LIN {X 0,Y 392.441,Z 295.362,A -85,B 0,C 180,E1 -11714.837,E2 -11714.837} C_VEL
LIN {X 0,Y 393.126,Z 283.476,A -85,B 0,C 180,E1 -11715.821,E2 -11715.821} C_VEL
LIN {X 0,Y 393.865,Z 270.295,A -85,B 0,C 180,E1 -11716.664,E2 -11716.664} C_VEL
LIN {X 0,Y 392.022,Z 258.735,A -85,B 0,C 180,E1 -11717.291,E2 -11717.291} C_VEL
LIN {X 0,Y 389.995,Z 247.385,A -85,B 0,C 180,E1 -11717.777,E2 -11717.777} C_VEL
LIN {X 0,Y 390.225,Z 238.96,A -85,B 0,C 180,E1 -11721.113,E2 -11721.113} C_VEL
LIN {X 0,Y 390.437,Z 231.991,A -85,B 0,C 180,E1 -11723.891,E2 -11723.891} C_VEL
LIN {X 0,Y 390.676,Z 223.459,A -85,B 0,C 180,E1 -11727.305,E2 -11727.305} C_VEL
LIN {X 0,Y 391.018,Z 214.714,A -85,B 0,C 180,E1 -11730.825,E2 -11730.825} C_VEL
LIN {X 0,Y 391.238,Z 206.117,A -85,B 0,C 180,E1 -11734.276,E2 -11734.276} C_VEL
LIN {X 0,Y 391.129,Z 201.01,A -85,B 0,C 180,E1 -11736.368,E2 -11736.368} C_VEL
LIN {X 0,Y 390.133,Z 194.889,A -85,B 0,C 180,E1 -11739.004,E2 -11739.004} C_VEL
LIN {X 0,Y 390.044,Z 194.901,A -85,B 0,C 180,E1 -11742.373,E2 -11742.373} C_VEL
LIN {X 0,Y 390.049,Z 194.896,A -85,B 0,C 180,E1 -11745.354,E2 -11745.354} C_VEL
LIN {X 0,Y 390.036,Z 194.901,A -85,B 0,C 180,E1 -11748.186,E2 -11748.186} C_VEL
LIN {X 0,Y 390.07,Z 194.899,A -85,B 0,C 180,E1 -11750.904,E2 -11750.904} C_VEL
LIN {X 0,Y 390.073,Z 194.899,A -85,B 0,C 180,E1 -11754.791,E2 -11754.791} C_VEL
LIN {X 0,Y 390.025,Z 194.903,A -85,B 0,C 180,E1 -11757.878,E2 -11757.878} C_VEL
LIN {X 0,Y 389.947,Z 194.914,A -85,B 0,C 180,E1 -11759.895,E2 -11759.895} C_VEL
LIN {X 0,Y 389.913,Z 195.341,A -85,B 0,C 180,E1 -11760.877,E2 -11760.877} C_VEL
LIN {X 0,Y 389.906,Z 199.409,A -85,B 0,C 180,E1 -11764.366,E2 -11764.366} C_VEL
LIN {X 0,Y 389.783,Z 203.49,A -85,B 0,C 180,E1 -11767.749,E2 -11767.749} C_VEL
LIN {X 0,Y 389.715,Z 207.645,A -85,B 0,C 180,E1 -11771.057,E2 -11771.057} C_VEL
LIN {X 0,Y 389.681,Z 211.96,A -85,B 0,C 180,E1 -11774.303,E2 -11774.303} C_VEL
LIN {X 0,Y 389.761,Z 217.229,A -85,B 0,C 180,E1 -11777.965,E2 -11777.965} C_VEL
LIN {X 0,Y 392.368,Z 228.553,A -85,B 0,C 180,E1 -11778.57,E2 -11778.57} C_VEL
LIN {X 0,Y 393.371,Z 233.68,A -85,B 0,C 180,E1 -11778.926,E2 -11778.926} C_VEL
LIN {X 0,Y 393.133,Z 243.41,A -85,B 0,C 180,E1 -11779.701,E2 -11779.701} C_VEL
LIN {X 0,Y 392.736,Z 250.958,A -85,B 0,C 180,E1 -11780.516,E2 -11780.516} C_VEL
LIN {X 0,Y 392.364,Z 256.371,A -85,B 0,C 180,E1 -11781.241,E2 -11781.241} C_VEL
LIN {X 0,Y 391.909,Z 262.54,A -85,B 0,C 180,E1 -11782.269,E2 -11782.269} C_VEL
LIN {X 0,Y 391.395,Z 268.341,A -85,B 0,C 180,E1 -11783.555,E2 -11783.555} C_VEL
LIN {X 0,Y 391.078,Z 272.615,A -85,B 0,C 180,E1 -11784.843,E2 -11784.843} C_VEL
LIN {X 0,Y 390.802,Z 275.178,A -85,B 0,C 180,E1 -11785.874,E2 -11785.874} C_VEL
LIN {X 0,Y 390.417,Z 277.099,A -85,B 0,C 180,E1 -11786.903,E2 -11786.903} C_VEL
LIN {X 0,Y 390.359,Z 278.393,A -85,B 0,C 180,E1 -11787.935,E2 -11787.935} C_VEL
LIN {X 0,Y 390.23,Z 279.168,A -85,B 0,C 180,E1 -11788.967,E2 -11788.967} C_VEL
LIN {X 0,Y 390.176,Z 279.434,A -85,B 0,C 180,E1 -11789.999,E2 -11789.999} C_VEL
LIN {X 0,Y 390.225,Z 279.209,A -85,B 0,C 180,E1 -11791.031,E2 -11791.031} C_VEL
LIN {X 0,Y 390.346,Z 278.488,A -85,B 0,C 180,E1 -11792.062,E2 -11792.062} C_VEL
LIN {X 0,Y 390.412,Z 277.251,A -85,B 0,C 180,E1 -11793.094,E2 -11793.094} C_VEL
LIN {X 0,Y 390.993,Z 274.224,A -85,B 0,C 180,E1 -11794.638,E2 -11794.638} C_VEL
LIN {X 0,Y 391.149,Z 269.687,A -85,B 0,C 180,E1 -11796.187,E2 -11796.187} C_VEL
LIN {X 0,Y 391.589,Z 266.668,A -85,B 0,C 180,E1 -11796.957,E2 -11796.957} C_VEL
LIN {X 0,Y 391.858,Z 262.997,A -85,B 0,C 180,E1 -11797.729,E2 -11797.729} C_VEL
LIN {X 0,Y 392.281,Z 257.796,A -85,B 0,C 180,E1 -11798.638,E2 -11798.638} C_VEL
LIN {X 0,Y 392.719,Z 251.934,A -85,B 0,C 180,E1 -11799.46,E2 -11799.46} C_VEL
LIN {X 0,Y 392.996,Z 245.724,A -85,B 0,C 180,E1 -11800.165,E2 -11800.165} C_VEL
LIN {X 0,Y 393.411,Z 237.435,A -85,B 0,C 180,E1 -11800.901,E2 -11800.901} C_VEL
LIN {X 0,Y 393.293,Z 232.95,A -85,B 0,C 180,E1 -11801.227,E2 -11801.227} C_VEL
LIN {X 0,Y 391.615,Z 228.223,A -85,B 0,C 180,E1 -11801.632,E2 -11801.632} C_VEL
LIN {X 0,Y 388.24,Z 222.83,A -85,B 0,C 180,E1 -11802.267,E2 -11802.267} C_VEL
LIN {X 0,Y 384.867,Z 218.57,A -85,B 0,C 180,E1 -11803.042,E2 -11803.042} C_VEL
LIN {X 0,Y 383.099,Z 216.211,A -85,B 0,C 180,E1 -11803.745,E2 -11803.745} C_VEL
LIN {X 0,Y 382.664,Z 215.17,A -85,B 0,C 180,E1 -11804.269,E2 -11804.269} C_VEL
LIN {X 0,Y 382.713,Z 211.016,A -85,B 0,C 180,E1 -11807.27,E2 -11807.27} C_VEL
LIN {X 0,Y 382.734,Z 206.813,A -85,B 0,C 180,E1 -11810.528,E2 -11810.528} C_VEL
LIN {X 0,Y 382.798,Z 202.837,A -85,B 0,C 180,E1 -11813.821,E2 -11813.821} C_VEL
LIN {X 0,Y 382.902,Z 198.648,A -85,B 0,C 180,E1 -11817.312,E2 -11817.312} C_VEL
LIN {X 0,Y 382.853,Z 195.894,A -85,B 0,C 180,E1 -11819.71,E2 -11819.71} C_VEL
LIN {X 0,Y 382.976,Z 195.779,A -85,B 0,C 180,E1 -11822.419,E2 -11822.419} C_VEL
LIN {X 0,Y 383.022,Z 195.774,A -85,B 0,C 180,E1 -11825.954,E2 -11825.954} C_VEL
LIN {X 0,Y 383.01,Z 195.776,A -85,B 0,C 180,E1 -11829.585,E2 -11829.585} C_VEL
LIN {X 0,Y 382.999,Z 195.778,A -85,B 0,C 180,E1 -11832.777,E2 -11832.777} C_VEL
LIN {X 0,Y 382.991,Z 195.776,A -85,B 0,C 180,E1 -11835.788,E2 -11835.788} C_VEL
LIN {X 0,Y 382.982,Z 195.779,A -85,B 0,C 180,E1 -11838.794,E2 -11838.794} C_VEL
LIN {X 0,Y 382.994,Z 195.776,A -85,B 0,C 180,E1 -11842.094,E2 -11842.094} C_VEL
LIN {X 0,Y 383.01,Z 195.772,A -85,B 0,C 180,E1 -11845.331,E2 -11845.331} C_VEL
LIN {X 0,Y 383.028,Z 195.771,A -85,B 0,C 180,E1 -11847.852,E2 -11847.852} C_VEL
LIN {X 0,Y 383.054,Z 195.766,A -85,B 0,C 180,E1 -11851.719,E2 -11851.719} C_VEL
LIN {X 0,Y 383.042,Z 195.762,A -85,B 0,C 180,E1 -11855.039,E2 -11855.039} C_VEL
LIN {X 0,Y 382.983,Z 195.775,A -85,B 0,C 180,E1 -11858.468,E2 -11858.468} C_VEL
LIN {X 0,Y 383.079,Z 195.769,A -85,B 0,C 180,E1 -11861.827,E2 -11861.827} C_VEL
LIN {X 0,Y 383.102,Z 195.754,A -85,B 0,C 180,E1 -11865.118,E2 -11865.118} C_VEL
LIN {X 0,Y 383.087,Z 195.762,A -85,B 0,C 180,E1 -11868.358,E2 -11868.358} C_VEL
LIN {X 0,Y 383.252,Z 195.743,A -85,B 0,C 180,E1 -11871.976,E2 -11871.976} C_VEL
LIN {X 0,Y 383.185,Z 195.747,A -85,B 0,C 180,E1 -11874.738,E2 -11874.738} C_VEL
LIN {X 0,Y 383.376,Z 195.727,A -85,B 0,C 180,E1 -11877.899,E2 -11877.899} C_VEL
LIN {X 0,Y 383.507,Z 195.702,A -85,B 0,C 180,E1 -11880,E2 -11880} C_VEL
LIN {X 0,Y 383.231,Z 195.746,A -85,B 0,C 180,E1 -11883.154,E2 -11883.154} C_VEL
LIN {X 0,Y 383.272,Z 195.74,A -85,B 0,C 180,E1 -11886.316,E2 -11886.316} C_VEL
LIN {X 0,Y 383.248,Z 195.744,A -85,B 0,C 180,E1 -11888.436,E2 -11888.436} C_VEL
LIN {X 0,Y 383.124,Z 195.756,A -85,B 0,C 180,E1 -11892.716,E2 -11892.716} C_VEL
LIN {X 0,Y 383.069,Z 195.77,A -85,B 0,C 180,E1 -11895.974,E2 -11895.974} C_VEL
LIN {X 0,Y 383.047,Z 195.77,A -85,B 0,C 180,E1 -11899.284,E2 -11899.284} C_VEL
LIN {X 0,Y 382.977,Z 195.78,A -85,B 0,C 180,E1 -11902.667,E2 -11902.667} C_VEL
LIN {X 0,Y 382.971,Z 195.783,A -85,B 0,C 180,E1 -11906.131,E2 -11906.131} C_VEL
LIN {X 0,Y 382.965,Z 195.784,A -85,B 0,C 180,E1 -11909.702,E2 -11909.702} C_VEL
LIN {X 0,Y 382.993,Z 195.78,A -85,B 0,C 180,E1 -11913.402,E2 -11913.402} C_VEL
LIN {X 0,Y 383.021,Z 195.774,A -85,B 0,C 180,E1 -11916.165,E2 -11916.165} C_VEL
LIN {X 0,Y 382.967,Z 195.773,A -85,B 0,C 180,E1 -11919.964,E2 -11919.964} C_VEL
LIN {X 0,Y 382.997,Z 195.782,A -85,B 0,C 180,E1 -11922.78,E2 -11922.78} C_VEL
LIN {X 0,Y 382.99,Z 195.778,A -85,B 0,C 180,E1 -11925.791,E2 -11925.791} C_VEL
LIN {X 0,Y 383.02,Z 195.777,A -85,B 0,C 180,E1 -11929.572,E2 -11929.572} C_VEL
LIN {X 0,Y 384.924,Z 203.825,A -85,B 0,C 180,E1 -11932.293,E2 -11932.293} C_VEL
LIN {X 0,Y 387.231,Z 213.656,A -85,B 0,C 180,E1 -11935.321,E2 -11935.321} C_VEL
LIN {X 0,Y 389.234,Z 223.254,A -85,B 0,C 180,E1 -11938.063,E2 -11938.063} C_VEL
LIN {X 0,Y 389.391,Z 225.849,A -85,B 0,C 180,E1 -11938.743,E2 -11938.743} C_VEL
LIN {X 0,Y 387.181,Z 241.285,A -85,B 0,C 180,E1 -11942.488,E2 -11942.488} C_VEL
LIN {X 0,Y 385.301,Z 257.405,A -85,B 0,C 180,E1 -11946.343,E2 -11946.343} C_VEL
LIN {X 0,Y 383.784,Z 273.332,A -85,B 0,C 180,E1 -11950.199,E2 -11950.199} C_VEL
LIN {X 0,Y 383.267,Z 280.554,A -85,B 0,C 180,E1 -11951.977,E2 -11951.977} C_VEL
LIN {X 0,Y 385,Z 300.047,A -85,B 0,C 180,E1 -11952.636,E2 -11952.636} C_VEL
LIN {X 0,Y 385.65,Z 311.521,A -85,B 0,C 180,E1 -11953.185,E2 -11953.185} C_VEL
LIN {X 0,Y 385.742,Z 319.562,A -85,B 0,C 180,E1 -11953.666,E2 -11953.666} C_VEL
LIN {X 0,Y 384.928,Z 331.35,A -85,B 0,C 180,E1 -11954.514,E2 -11954.514} C_VEL
LIN {X 0,Y 384.273,Z 342.675,A -85,B 0,C 180,E1 -11955.559,E2 -11955.559} C_VEL
LIN {X 0,Y 383.547,Z 353.146,A -85,B 0,C 180,E1 -11956.761,E2 -11956.761} C_VEL
LIN {X 0,Y 382.946,Z 362.582,A -85,B 0,C 180,E1 -11958.086,E2 -11958.086} C_VEL
LIN {X 0,Y 382.337,Z 371.679,A -85,B 0,C 180,E1 -11959.677,E2 -11959.677} C_VEL
LIN {X 0,Y 382.054,Z 379.013,A -85,B 0,C 180,E1 -11961.272,E2 -11961.272} C_VEL
LIN {X 0,Y 381.91,Z 383.943,A -85,B 0,C 180,E1 -11962.6,E2 -11962.6} C_VEL
LIN {X 0,Y 381.775,Z 388.418,A -85,B 0,C 180,E1 -11964.093,E2 -11964.093} C_VEL
LIN {X 0,Y 381.786,Z 392.244,A -85,B 0,C 180,E1 -11965.779,E2 -11965.779} C_VEL
LIN {X 0,Y 381.861,Z 394.015,A -85,B 0,C 180,E1 -11966.836,E2 -11966.836} C_VEL
LIN {X 0,Y 381.878,Z 395.313,A -85,B 0,C 180,E1 -11967.892,E2 -11967.892} C_VEL
LIN {X 0,Y 381.878,Z 396.187,A -85,B 0,C 180,E1 -11968.947,E2 -11968.947} C_VEL
LIN {X 0,Y 381.914,Z 396.626,A -85,B 0,C 180,E1 -11970.001,E2 -11970.001} C_VEL
LIN {X 0,Y 381.857,Z 396.594,A -85,B 0,C 180,E1 -11971.056,E2 -11971.056} C_VEL
LIN {X 0,Y 381.866,Z 396.15,A -85,B 0,C 180,E1 -11972.111,E2 -11972.111} C_VEL
LIN {X 0,Y 381.779,Z 395.289,A -85,B 0,C 180,E1 -11973.167,E2 -11973.167} C_VEL
LIN {X 0,Y 381.77,Z 393.964,A -85,B 0,C 180,E1 -11974.224,E2 -11974.224} C_VEL
LIN {X 0,Y 381.77,Z 390.247,A -85,B 0,C 180,E1 -11976.233,E2 -11976.233} C_VEL
LIN {X 0,Y 381.983,Z 385.806,A -85,B 0,C 180,E1 -11977.933,E2 -11977.933} C_VEL
LIN {X 0,Y 382.401,Z 379.388,A -85,B 0,C 180,E1 -11979.789,E2 -11979.789} C_VEL
LIN {X 0,Y 382.931,Z 372.469,A -85,B 0,C 180,E1 -11981.38,E2 -11981.38} C_VEL
LIN {X 0,Y 383.876,Z 364.003,A -85,B 0,C 180,E1 -11982.961,E2 -11982.961} C_VEL
LIN {X 0,Y 384.806,Z 353.59,A -85,B 0,C 180,E1 -11984.538,E2 -11984.538} C_VEL
LIN {X 0,Y 386.105,Z 342.845,A -85,B 0,C 180,E1 -11985.846,E2 -11985.846} C_VEL
LIN {X 0,Y 387.472,Z 330.997,A -85,B 0,C 180,E1 -11987.008,E2 -11987.008} C_VEL
LIN {X 0,Y 388.687,Z 318.195,A -85,B 0,C 180,E1 -11988.011,E2 -11988.011} C_VEL
LIN {X 0,Y 388.737,Z 304.837,A -85,B 0,C 180,E1 -11988.892,E2 -11988.892} C_VEL
LIN {X 0,Y 387.598,Z 290.655,A -85,B 0,C 180,E1 -11989.68,E2 -11989.68} C_VEL
LIN {X 0,Y 385.077,Z 275.775,A -85,B 0,C 180,E1 -11990.475,E2 -11990.475} C_VEL
LIN {X 0,Y 384.394,Z 266.537,A -85,B 0,C 180,E1 -11991.45,E2 -11991.45} C_VEL
LIN {X 0,Y 386.367,Z 248.038,A -85,B 0,C 180,E1 -11995.886,E2 -11995.886} C_VEL
LIN {X 0,Y 388.604,Z 230.925,A -85,B 0,C 180,E1 -11999.996,E2 -11999.996} C_VEL
LIN {X 0,Y 389.414,Z 224.596,A -85,B 0,C 180,E1 -12001.561,E2 -12001.561} C_VEL
LIN {X 0,Y 387.476,Z 215.101,A -85,B 0,C 180,E1 -12004.214,E2 -12004.214} C_VEL
LIN {X 0,Y 385.15,Z 204.861,A -85,B 0,C 180,E1 -12007.354,E2 -12007.354} C_VEL
LIN {X 0,Y 384.083,Z 200.232,A -85,B 0,C 180,E1 -12008.887,E2 -12008.887} C_VEL
LIN {X 0,Y 384.548,Z 199.877,A -85,B 0,C 180,E1 -12009.862,E2 -12009.862} C_VEL
LIN {X 0,Y 384.84,Z 201.165,A -85,B 0,C 180,E1 -12013.073,E2 -12013.073} C_VEL
LIN {X 0,Y 385.222,Z 202.398,A -85,B 0,C 180,E1 -12014.641,E2 -12014.641} C_VEL
LIN {X 0,Y 386.114,Z 205.789,A -85,B 0,C 180,E1 -12017.665,E2 -12017.665} C_VEL
LIN {X 0,Y 387.063,Z 210.04,A -85,B 0,C 180,E1 -12020.543,E2 -12020.543} C_VEL
LIN {X 0,Y 387.815,Z 214.746,A -85,B 0,C 180,E1 -12023.271,E2 -12023.271} C_VEL
LIN {X 0,Y 387.943,Z 217.442,A -85,B 0,C 180,E1 -12024.611,E2 -12024.611} C_VEL
LIN {X 0,Y 386.832,Z 225.39,A -85,B 0,C 180,E1 -12028.205,E2 -12028.205} C_VEL
LIN {X 0,Y 386.084,Z 233.594,A -85,B 0,C 180,E1 -12031.752,E2 -12031.752} C_VEL
LIN {X 0,Y 385.508,Z 241.602,A -85,B 0,C 180,E1 -12035.209,E2 -12035.209} C_VEL
LIN {X 0,Y 384.943,Z 249.614,A -85,B 0,C 180,E1 -12038.612,E2 -12038.612} C_VEL
LIN {X 0,Y 384.852,Z 252.197,A -85,B 0,C 180,E1 -12039.664,E2 -12039.664} C_VEL
LIN {X 0,Y 389.3,Z 265.874,A -85,B 0,C 180,E1 -12040.724,E2 -12040.724} C_VEL
LIN {X 0,Y 391.121,Z 274.403,A -85,B 0,C 180,E1 -12041.405,E2 -12041.405} C_VEL
LIN {X 0,Y 390.072,Z 287.025,A -85,B 0,C 180,E1 -12042.3,E2 -12042.3} C_VEL
LIN {X 0,Y 388.872,Z 298.96,A -85,B 0,C 180,E1 -12043.372,E2 -12043.372} C_VEL
LIN {X 0,Y 387.61,Z 310.068,A -85,B 0,C 180,E1 -12044.623,E2 -12044.623} C_VEL
LIN {X 0,Y 386.508,Z 318.618,A -85,B 0,C 180,E1 -12045.79,E2 -12045.79} C_VEL
LIN {X 0,Y 385.488,Z 326.598,A -85,B 0,C 180,E1 -12047.095,E2 -12047.095} C_VEL
LIN {X 0,Y 384.521,Z 334.416,A -85,B 0,C 180,E1 -12048.669,E2 -12048.669} C_VEL
LIN {X 0,Y 383.62,Z 341.722,A -85,B 0,C 180,E1 -12050.51,E2 -12050.51} C_VEL
LIN {X 0,Y 382.899,Z 347.344,A -85,B 0,C 180,E1 -12052.38,E2 -12052.38} C_VEL
LIN {X 0,Y 382.407,Z 350.368,A -85,B 0,C 180,E1 -12053.669,E2 -12053.669} C_VEL
LIN {X 0,Y 382.386,Z 352.255,A -85,B 0,C 180,E1 -12054.727,E2 -12054.727} C_VEL
LIN {X 0,Y 382.246,Z 353.747,A -85,B 0,C 180,E1 -12055.782,E2 -12055.782} C_VEL
LIN {X 0,Y 382.043,Z 354.843,A -85,B 0,C 180,E1 -12056.836,E2 -12056.836} C_VEL
LIN {X 0,Y 381.887,Z 355.487,A -85,B 0,C 180,E1 -12057.891,E2 -12057.891} C_VEL
LIN {X 0,Y 381.777,Z 355.73,A -85,B 0,C 180,E1 -12058.945,E2 -12058.945} C_VEL
LIN {X 0,Y 381.725,Z 355.576,A -85,B 0,C 180,E1 -12060,E2 -12060} C_VEL
LIN {X 0,Y 381.742,Z 354.991,A -85,B 0,C 180,E1 -12061.055,E2 -12061.055} C_VEL
LIN {X 0,Y 381.827,Z 353.971,A -85,B 0,C 180,E1 -12062.11,E2 -12062.11} C_VEL
LIN {X 0,Y 381.878,Z 352.553,A -85,B 0,C 180,E1 -12063.165,E2 -12063.165} C_VEL
LIN {X 0,Y 381.921,Z 349.589,A -85,B 0,C 180,E1 -12064.75,E2 -12064.75} C_VEL
LIN {X 0,Y 382.122,Z 345.564,A -85,B 0,C 180,E1 -12066.336,E2 -12066.336} C_VEL
LIN {X 0,Y 382.464,Z 339.365,A -85,B 0,C 180,E1 -12068.187,E2 -12068.187} C_VEL
LIN {X 0,Y 382.954,Z 332.597,A -85,B 0,C 180,E1 -12069.774,E2 -12069.774} C_VEL
LIN {X 0,Y 383.495,Z 324.224,A -85,B 0,C 180,E1 -12071.362,E2 -12071.362} C_VEL
LIN {X 0,Y 384.135,Z 315.655,A -85,B 0,C 180,E1 -12072.683,E2 -12072.683} C_VEL
LIN {X 0,Y 384.915,Z 304.334,A -85,B 0,C 180,E1 -12074.11,E2 -12074.11} C_VEL
LIN {X 0,Y 385.671,Z 292.196,A -85,B 0,C 180,E1 -12075.321,E2 -12075.321} C_VEL
LIN {X 0,Y 386.335,Z 280.59,A -85,B 0,C 180,E1 -12076.242,E2 -12076.242} C_VEL
LIN {X 0,Y 386.905,Z 270.133,A -85,B 0,C 180,E1 -12076.896,E2 -12076.896} C_VEL
LIN {X 0,Y 384.444,Z 255.949,A -85,B 0,C 180,E1 -12077.653,E2 -12077.653} C_VEL
LIN {X 0,Y 382.945,Z 247.664,A -85,B 0,C 180,E1 -12078.024,E2 -12078.024} C_VEL
LIN {X 0,Y 383.22,Z 238.902,A -85,B 0,C 180,E1 -12081.518,E2 -12081.518} C_VEL
LIN {X 0,Y 383.427,Z 231.838,A -85,B 0,C 180,E1 -12084.357,E2 -12084.357} C_VEL
LIN {X 0,Y 383.696,Z 223.209,A -85,B 0,C 180,E1 -12087.845,E2 -12087.845} C_VEL
LIN {X 0,Y 384.063,Z 214.34,A -85,B 0,C 180,E1 -12091.435,E2 -12091.435} C_VEL
LIN {X 0,Y 384.305,Z 205.172,A -85,B 0,C 180,E1 -12095.173,E2 -12095.173} C_VEL
LIN {X 0,Y 383.848,Z 200.338,A -85,B 0,C 180,E1 -12097.172,E2 -12097.172} C_VEL
LIN {X 0,Y 383.08,Z 195.768,A -85,B 0,C 180,E1 -12099.183,E2 -12099.183} C_VEL
LIN {X 0,Y 383.011,Z 195.778,A -85,B 0,C 180,E1 -12102.778,E2 -12102.778} C_VEL
LIN {X 0,Y 383.003,Z 195.777,A -85,B 0,C 180,E1 -12105.789,E2 -12105.789} C_VEL
LIN {X 0,Y 382.993,Z 195.78,A -85,B 0,C 180,E1 -12108.795,E2 -12108.795} C_VEL
LIN {X 0,Y 383,Z 195.781,A -85,B 0,C 180,E1 -12112.097,E2 -12112.097} C_VEL
LIN {X 0,Y 383.016,Z 195.779,A -85,B 0,C 180,E1 -12115.331,E2 -12115.331} C_VEL
LIN {X 0,Y 383.004,Z 195.778,A -85,B 0,C 180,E1 -12117.849,E2 -12117.849} C_VEL
LIN {X 0,Y 382.856,Z 195.798,A -85,B 0,C 180,E1 -12120.287,E2 -12120.287} C_VEL
LIN {X 0,Y 382.913,Z 198.525,A -85,B 0,C 180,E1 -12122.686,E2 -12122.686} C_VEL
LIN {X 0,Y 382.8,Z 202.65,A -85,B 0,C 180,E1 -12126.176,E2 -12126.176} C_VEL
LIN {X 0,Y 382.739,Z 206.829,A -85,B 0,C 180,E1 -12129.58,E2 -12129.58} C_VEL
LIN {X 0,Y 382.717,Z 211.112,A -85,B 0,C 180,E1 -12132.912,E2 -12132.912} C_VEL
LIN {X 0,Y 382.717,Z 216.426,A -85,B 0,C 180,E1 -12136.722,E2 -12136.722} C_VEL
LIN {X 0,Y 382.771,Z 218,A -85,B 0,C 180,E1 -12137.708,E2 -12137.708} C_VEL
LIN {X 0,Y 385.092,Z 227.759,A -85,B 0,C 180,E1 -12138.218,E2 -12138.218} C_VEL
LIN {X 0,Y 386.503,Z 235.079,A -85,B 0,C 180,E1 -12138.727,E2 -12138.727} C_VEL
LIN {X 0,Y 386.249,Z 244.611,A -85,B 0,C 180,E1 -12139.515,E2 -12139.515} C_VEL
LIN {X 0,Y 385.828,Z 252.004,A -85,B 0,C 180,E1 -12140.334,E2 -12140.334} C_VEL
LIN {X 0,Y 385.435,Z 257.447,A -85,B 0,C 180,E1 -12141.083,E2 -12141.083} C_VEL
LIN {X 0,Y 384.947,Z 263.581,A -85,B 0,C 180,E1 -12142.129,E2 -12142.129} C_VEL
LIN {X 0,Y 384.417,Z 269.356,A -85,B 0,C 180,E1 -12143.438,E2 -12143.438} C_VEL
LIN {X 0,Y 384.082,Z 273.607,A -85,B 0,C 180,E1 -12144.749,E2 -12144.749} C_VEL
LIN {X 0,Y 383.799,Z 276.161,A -85,B 0,C 180,E1 -12145.798,E2 -12145.798} C_VEL
LIN {X 0,Y 383.403,Z 278.077,A -85,B 0,C 180,E1 -12146.846,E2 -12146.846} C_VEL
LIN {X 0,Y 383.34,Z 279.368,A -85,B 0,C 180,E1 -12147.897,E2 -12147.897} C_VEL
LIN {X 0,Y 383.206,Z 280.142,A -85,B 0,C 180,E1 -12148.948,E2 -12148.948} C_VEL
LIN {X 0,Y 383.15,Z 280.407,A -85,B 0,C 180,E1 -12149.999,E2 -12149.999} C_VEL
LIN {X 0,Y 383.201,Z 280.182,A -85,B 0,C 180,E1 -12151.05,E2 -12151.05} C_VEL
LIN {X 0,Y 383.327,Z 279.462,A -85,B 0,C 180,E1 -12152.1,E2 -12152.1} C_VEL
LIN {X 0,Y 383.398,Z 278.228,A -85,B 0,C 180,E1 -12153.151,E2 -12153.151} C_VEL
LIN {X 0,Y 383.995,Z 275.209,A -85,B 0,C 180,E1 -12154.723,E2 -12154.723} C_VEL
LIN {X 0,Y 384.163,Z 270.69,A -85,B 0,C 180,E1 -12156.3,E2 -12156.3} C_VEL
LIN {X 0,Y 384.617,Z 267.684,A -85,B 0,C 180,E1 -12157.084,E2 -12157.084} C_VEL
LIN {X 0,Y 384.901,Z 264.035,A -85,B 0,C 180,E1 -12157.87,E2 -12157.87} C_VEL
LIN {X 0,Y 385.423,Z 258.095,A -85,B 0,C 180,E1 -12158.915,E2 -12158.915} C_VEL
LIN {X 0,Y 385.908,Z 251.406,A -85,B 0,C 180,E1 -12159.842,E2 -12159.842} C_VEL
LIN {X 0,Y 386.288,Z 242.955,A -85,B 0,C 180,E1 -12160.746,E2 -12160.746} C_VEL
LIN {X 0,Y 386.512,Z 234.664,A -85,B 0,C 180,E1 -12161.403,E2 -12161.403} C_VEL
LIN {X 0,Y 384.452,Z 224.93,A -85,B 0,C 180,E1 -12162.05,E2 -12162.05} C_VEL
LIN {X 0,Y 382.738,Z 217.845,A -85,B 0,C 180,E1 -12162.425,E2 -12162.425} C_VEL
LIN {X 0,Y 382.664,Z 215.17,A -85,B 0,C 180,E1 -12164.269,E2 -12164.269} C_VEL
LIN {X 0,Y 381.98,Z 214.053,A -85,B 0,C 180,E1 -12165.131,E2 -12165.131} C_VEL
LIN {X 0,Y 379.149,Z 212.545,A -85,B 0,C 180,E1 -12166.543,E2 -12166.543} C_VEL
LIN {X 0,Y 376.766,Z 211.369,A -85,B 0,C 180,E1 -12167.686,E2 -12167.686} C_VEL
LIN {X 0,Y 375.744,Z 210.371,A -85,B 0,C 180,E1 -12168.566,E2 -12168.566} C_VEL
LIN {X 0,Y 375.659,Z 210.002,A -85,B 0,C 180,E1 -12168.863,E2 -12168.863} C_VEL
LIN {X 0,Y 375.729,Z 206.127,A -85,B 0,C 180,E1 -12171.967,E2 -12171.967} C_VEL
LIN {X 0,Y 375.78,Z 203.339,A -85,B 0,C 180,E1 -12174.294,E2 -12174.294} C_VEL
LIN {X 0,Y 375.858,Z 200.519,A -85,B 0,C 180,E1 -12176.663,E2 -12176.663} C_VEL
LIN {X 0,Y 375.855,Z 197.709,A -85,B 0,C 180,E1 -12179.087,E2 -12179.087} C_VEL
LIN {X 0,Y 375.888,Z 196.664,A -85,B 0,C 180,E1 -12180.317,E2 -12180.317} C_VEL
LIN {X 0,Y 375.943,Z 196.656,A -85,B 0,C 180,E1 -12182.827,E2 -12182.827} C_VEL
LIN {X 0,Y 375.954,Z 196.657,A -85,B 0,C 180,E1 -12185.414,E2 -12185.414} C_VEL
LIN {X 0,Y 375.97,Z 196.652,A -85,B 0,C 180,E1 -12188.269,E2 -12188.269} C_VEL
LIN {X 0,Y 375.929,Z 196.657,A -85,B 0,C 180,E1 -12191.599,E2 -12191.599} C_VEL
LIN {X 0,Y 375.947,Z 196.657,A -85,B 0,C 180,E1 -12195.263,E2 -12195.263} C_VEL
LIN {X 0,Y 375.934,Z 196.654,A -85,B 0,C 180,E1 -12199.132,E2 -12199.132} C_VEL
LIN {X 0,Y 375.959,Z 196.652,A -85,B 0,C 180,E1 -12201.911,E2 -12201.911} C_VEL
LIN {X 0,Y 375.971,Z 196.649,A -85,B 0,C 180,E1 -12205.331,E2 -12205.331} C_VEL
LIN {X 0,Y 375.968,Z 196.656,A -85,B 0,C 180,E1 -12208.439,E2 -12208.439} C_VEL
LIN {X 0,Y 375.993,Z 196.65,A -85,B 0,C 180,E1 -12212.141,E2 -12212.141} C_VEL
LIN {X 0,Y 375.996,Z 196.641,A -85,B 0,C 180,E1 -12214.538,E2 -12214.538} C_VEL
LIN {X 0,Y 375.953,Z 196.654,A -85,B 0,C 180,E1 -12218.045,E2 -12218.045} C_VEL
LIN {X 0,Y 376.013,Z 196.645,A -85,B 0,C 180,E1 -12221.473,E2 -12221.473} C_VEL
LIN {X 0,Y 376.05,Z 196.632,A -85,B 0,C 180,E1 -12224.832,E2 -12224.832} C_VEL
LIN {X 0,Y 376.039,Z 196.641,A -85,B 0,C 180,E1 -12228.136,E2 -12228.136} C_VEL
LIN {X 0,Y 376.207,Z 196.621,A -85,B 0,C 180,E1 -12231.919,E2 -12231.919} C_VEL
LIN {X 0,Y 376.157,Z 196.623,A -85,B 0,C 180,E1 -12234.64,E2 -12234.64} C_VEL
LIN {X 0,Y 376.342,Z 196.603,A -85,B 0,C 180,E1 -12237.86,E2 -12237.86} C_VEL
LIN {X 0,Y 376.477,Z 196.578,A -85,B 0,C 180,E1 -12240,E2 -12240} C_VEL
LIN {X 0,Y 376.17,Z 196.625,A -85,B 0,C 180,E1 -12243.213,E2 -12243.213} C_VEL
LIN {X 0,Y 376.232,Z 196.618,A -85,B 0,C 180,E1 -12246.435,E2 -12246.435} C_VEL
LIN {X 0,Y 376.194,Z 196.62,A -85,B 0,C 180,E1 -12248.595,E2 -12248.595} C_VEL
LIN {X 0,Y 376.037,Z 196.644,A -85,B 0,C 180,E1 -12251.864,E2 -12251.864} C_VEL
LIN {X 0,Y 376.046,Z 196.642,A -85,B 0,C 180,E1 -12255.168,E2 -12255.168} C_VEL
LIN {X 0,Y 375.991,Z 196.651,A -85,B 0,C 180,E1 -12258.528,E2 -12258.528} C_VEL
LIN {X 0,Y 375.943,Z 196.659,A -85,B 0,C 180,E1 -12261.956,E2 -12261.956} C_VEL
LIN {X 0,Y 375.947,Z 196.658,A -85,B 0,C 180,E1 -12264.285,E2 -12264.285} C_VEL
LIN {X 0,Y 375.906,Z 196.663,A -85,B 0,C 180,E1 -12267.866,E2 -12267.866} C_VEL
LIN {X 0,Y 375.947,Z 196.659,A -85,B 0,C 180,E1 -12271.563,E2 -12271.563} C_VEL
LIN {X 0,Y 375.947,Z 196.656,A -85,B 0,C 180,E1 -12275.417,E2 -12275.417} C_VEL
LIN {X 0,Y 375.927,Z 196.66,A -85,B 0,C 180,E1 -12278.264,E2 -12278.264} C_VEL
LIN {X 0,Y 375.911,Z 196.653,A -85,B 0,C 180,E1 -12281.599,E2 -12281.599} C_VEL
LIN {X 0,Y 375.919,Z 196.662,A -85,B 0,C 180,E1 -12284.733,E2 -12284.733} C_VEL
LIN {X 0,Y 375.927,Z 196.649,A -85,B 0,C 180,E1 -12288.401,E2 -12288.401} C_VEL
LIN {X 0,Y 375.972,Z 196.823,A -85,B 0,C 180,E1 -12289.065,E2 -12289.065} C_VEL
LIN {X 0,Y 377.751,Z 204.13,A -85,B 0,C 180,E1 -12291.622,E2 -12291.622} C_VEL
LIN {X 0,Y 380.267,Z 214.887,A -85,B 0,C 180,E1 -12295.047,E2 -12295.047} C_VEL
LIN {X 0,Y 382.452,Z 225.437,A -85,B 0,C 180,E1 -12298.11,E2 -12298.11} C_VEL
LIN {X 0,Y 382.237,Z 228.933,A -85,B 0,C 180,E1 -12299.016,E2 -12299.016} C_VEL
LIN {X 0,Y 379.837,Z 245.163,A -85,B 0,C 180,E1 -12303.046,E2 -12303.046} C_VEL
LIN {X 0,Y 378.066,Z 260.186,A -85,B 0,C 180,E1 -12306.734,E2 -12306.734} C_VEL
LIN {X 0,Y 376.56,Z 275.877,A -85,B 0,C 180,E1 -12310.655,E2 -12310.655} C_VEL
LIN {X 0,Y 376.226,Z 280.307,A -85,B 0,C 180,E1 -12311.74,E2 -12311.74} C_VEL
LIN {X 0,Y 377.957,Z 299.837,A -85,B 0,C 180,E1 -12312.42,E2 -12312.42} C_VEL
LIN {X 0,Y 378.62,Z 310.331,A -85,B 0,C 180,E1 -12312.933,E2 -12312.933} C_VEL
LIN {X 0,Y 378.752,Z 319.578,A -85,B 0,C 180,E1 -12313.495,E2 -12313.495} C_VEL
LIN {X 0,Y 377.919,Z 331.247,A -85,B 0,C 180,E1 -12314.358,E2 -12314.358} C_VEL
LIN {X 0,Y 377.186,Z 343.103,A -85,B 0,C 180,E1 -12315.488,E2 -12315.488} C_VEL
LIN {X 0,Y 376.456,Z 353.958,A -85,B 0,C 180,E1 -12316.781,E2 -12316.781} C_VEL
LIN {X 0,Y 375.826,Z 363.128,A -85,B 0,C 180,E1 -12318.131,E2 -12318.131} C_VEL
LIN {X 0,Y 375.234,Z 372.052,A -85,B 0,C 180,E1 -12319.752,E2 -12319.752} C_VEL
LIN {X 0,Y 374.961,Z 379.235,A -85,B 0,C 180,E1 -12321.378,E2 -12321.378} C_VEL
LIN {X 0,Y 374.79,Z 384.907,A -85,B 0,C 180,E1 -12323,E2 -12323} C_VEL
LIN {X 0,Y 374.758,Z 389.321,A -85,B 0,C 180,E1 -12324.621,E2 -12324.621} C_VEL
LIN {X 0,Y 374.715,Z 391.618,A -85,B 0,C 180,E1 -12325.699,E2 -12325.699} C_VEL
LIN {X 0,Y 374.765,Z 393.455,A -85,B 0,C 180,E1 -12326.776,E2 -12326.776} C_VEL
LIN {X 0,Y 374.809,Z 394.788,A -85,B 0,C 180,E1 -12327.852,E2 -12327.852} C_VEL
LIN {X 0,Y 374.801,Z 395.694,A -85,B 0,C 180,E1 -12328.927,E2 -12328.927} C_VEL
LIN {X 0,Y 374.833,Z 396.183,A -85,B 0,C 180,E1 -12330.001,E2 -12330.001} C_VEL
LIN {X 0,Y 374.782,Z 396.198,A -85,B 0,C 180,E1 -12331.076,E2 -12331.076} C_VEL
LIN {X 0,Y 374.794,Z 395.786,A -85,B 0,C 180,E1 -12332.151,E2 -12332.151} C_VEL
LIN {X 0,Y 374.679,Z 394.954,A -85,B 0,C 180,E1 -12333.227,E2 -12333.227} C_VEL
LIN {X 0,Y 374.689,Z 393.696,A -85,B 0,C 180,E1 -12334.304,E2 -12334.304} C_VEL
LIN {X 0,Y 374.688,Z 390.342,A -85,B 0,C 180,E1 -12336.216,E2 -12336.216} C_VEL
LIN {X 0,Y 374.91,Z 385.686,A -85,B 0,C 180,E1 -12338.084,E2 -12338.084} C_VEL
LIN {X 0,Y 375.371,Z 379.412,A -85,B 0,C 180,E1 -12339.974,E2 -12339.974} C_VEL
LIN {X 0,Y 376.098,Z 371.346,A -85,B 0,C 180,E1 -12341.863,E2 -12341.863} C_VEL
LIN {X 0,Y 376.956,Z 364.291,A -85,B 0,C 180,E1 -12343.204,E2 -12343.204} C_VEL
LIN {X 0,Y 377.903,Z 354.57,A -85,B 0,C 180,E1 -12344.745,E2 -12344.745} C_VEL
LIN {X 0,Y 379.337,Z 343.648,A -85,B 0,C 180,E1 -12346.137,E2 -12346.137} C_VEL
LIN {X 0,Y 380.764,Z 332.213,A -85,B 0,C 180,E1 -12347.317,E2 -12347.317} C_VEL
LIN {X 0,Y 382.124,Z 319.753,A -85,B 0,C 180,E1 -12348.347,E2 -12348.347} C_VEL
LIN {X 0,Y 382.388,Z 307.435,A -85,B 0,C 180,E1 -12349.218,E2 -12349.218} C_VEL
LIN {X 0,Y 381.453,Z 292.78,A -85,B 0,C 180,E1 -12350.104,E2 -12350.104} C_VEL
LIN {X 0,Y 379.099,Z 278.124,A -85,B 0,C 180,E1 -12350.926,E2 -12350.926} C_VEL
LIN {X 0,Y 378.518,Z 275.536,A -85,B 0,C 180,E1 -12351.09,E2 -12351.09} C_VEL
LIN {X 0,Y 377.757,Z 263.252,A -85,B 0,C 180,E1 -12352.493,E2 -12352.493} C_VEL
LIN {X 0,Y 379.708,Z 246.268,A -85,B 0,C 180,E1 -12356.669,E2 -12356.669} C_VEL
LIN {X 0,Y 382.237,Z 228.809,A -85,B 0,C 180,E1 -12360.987,E2 -12360.987} C_VEL
LIN {X 0,Y 382.43,Z 225.324,A -85,B 0,C 180,E1 -12361.895,E2 -12361.895} C_VEL
LIN {X 0,Y 380.241,Z 214.793,A -85,B 0,C 180,E1 -12364.959,E2 -12364.959} C_VEL
LIN {X 0,Y 377.981,Z 205.17,A -85,B 0,C 180,E1 -12368.034,E2 -12368.034} C_VEL
LIN {X 0,Y 378.508,Z 204.372,A -85,B 0,C 180,E1 -12369.147,E2 -12369.147} C_VEL
LIN {X 0,Y 378.75,Z 204.167,A -85,B 0,C 180,E1 -12370.502,E2 -12370.502} C_VEL
LIN {X 0,Y 379.122,Z 205.478,A -85,B 0,C 180,E1 -12373.7,E2 -12373.7} C_VEL
LIN {X 0,Y 379.726,Z 208.272,A -85,B 0,C 180,E1 -12376.78,E2 -12376.78} C_VEL
LIN {X 0,Y 380.532,Z 212.074,A -85,B 0,C 180,E1 -12379.728,E2 -12379.728} C_VEL
LIN {X 0,Y 381.22,Z 216.443,A -85,B 0,C 180,E1 -12382.528,E2 -12382.528} C_VEL
LIN {X 0,Y 381.415,Z 219.89,A -85,B 0,C 180,E1 -12384.422,E2 -12384.422} C_VEL
LIN {X 0,Y 380.365,Z 226.847,A -85,B 0,C 180,E1 -12387.6,E2 -12387.6} C_VEL
LIN {X 0,Y 379.507,Z 234.843,A -85,B 0,C 180,E1 -12391.217,E2 -12391.217} C_VEL
LIN {X 0,Y 378.684,Z 244.361,A -85,B 0,C 180,E1 -12395.423,E2 -12395.423} C_VEL
LIN {X 0,Y 378.064,Z 252.663,A -85,B 0,C 180,E1 -12399.015,E2 -12399.015} C_VEL
LIN {X 0,Y 382.423,Z 265.485,A -85,B 0,C 180,E1 -12400.085,E2 -12400.085} C_VEL
LIN {X 0,Y 384.688,Z 275.647,A -85,B 0,C 180,E1 -12400.948,E2 -12400.948} C_VEL
LIN {X 0,Y 384.441,Z 280.567,A -85,B 0,C 180,E1 -12401.295,E2 -12401.295} C_VEL
LIN {X 0,Y 383.202,Z 292.877,A -85,B 0,C 180,E1 -12402.289,E2 -12402.289} C_VEL
LIN {X 0,Y 381.906,Z 303.782,A -85,B 0,C 180,E1 -12403.381,E2 -12403.381} C_VEL
LIN {X 0,Y 380.486,Z 314.649,A -85,B 0,C 180,E1 -12404.739,E2 -12404.739} C_VEL
LIN {X 0,Y 379.253,Z 323.345,A -85,B 0,C 180,E1 -12406.06,E2 -12406.06} C_VEL
LIN {X 0,Y 378.073,Z 331.855,A -85,B 0,C 180,E1 -12407.656,E2 -12407.656} C_VEL
LIN {X 0,Y 377.239,Z 338.755,A -85,B 0,C 180,E1 -12409.263,E2 -12409.263} C_VEL
LIN {X 0,Y 376.426,Z 344.339,A -85,B 0,C 180,E1 -12410.869,E2 -12410.869} C_VEL
LIN {X 0,Y 375.852,Z 348.728,A -85,B 0,C 180,E1 -12412.479,E2 -12412.479} C_VEL
LIN {X 0,Y 375.39,Z 351.06,A -85,B 0,C 180,E1 -12413.55,E2 -12413.55} C_VEL
LIN {X 0,Y 375.339,Z 352.898,A -85,B 0,C 180,E1 -12414.628,E2 -12414.628} C_VEL
LIN {X 0,Y 375.207,Z 354.342,A -85,B 0,C 180,E1 -12415.703,E2 -12415.703} C_VEL
LIN {X 0,Y 374.993,Z 355.372,A -85,B 0,C 180,E1 -12416.777,E2 -12416.777} C_VEL
LIN {X 0,Y 374.824,Z 355.966,A -85,B 0,C 180,E1 -12417.851,E2 -12417.851} C_VEL
LIN {X 0,Y 374.708,Z 356.167,A -85,B 0,C 180,E1 -12418.925,E2 -12418.925} C_VEL
LIN {X 0,Y 374.655,Z 355.964,A -85,B 0,C 180,E1 -12420,E2 -12420} C_VEL
LIN {X 0,Y 374.674,Z 355.308,A -85,B 0,C 180,E1 -12421.075,E2 -12421.075} C_VEL
LIN {X 0,Y 374.746,Z 354.246,A -85,B 0,C 180,E1 -12422.15,E2 -12422.15} C_VEL
LIN {X 0,Y 374.783,Z 352.785,A -85,B 0,C 180,E1 -12423.225,E2 -12423.225} C_VEL
LIN {X 0,Y 374.86,Z 349.734,A -85,B 0,C 180,E1 -12424.84,E2 -12424.84} C_VEL
LIN {X 0,Y 375.092,Z 344.712,A -85,B 0,C 180,E1 -12426.753,E2 -12426.753} C_VEL
LIN {X 0,Y 375.471,Z 338.254,A -85,B 0,C 180,E1 -12428.612,E2 -12428.612} C_VEL
LIN {X 0,Y 375.984,Z 331.113,A -85,B 0,C 180,E1 -12430.229,E2 -12430.229} C_VEL
LIN {X 0,Y 376.587,Z 322.251,A -85,B 0,C 180,E1 -12431.846,E2 -12431.846} C_VEL
LIN {X 0,Y 377.411,Z 312.233,A -85,B 0,C 180,E1 -12433.323,E2 -12433.323} C_VEL
LIN {X 0,Y 378.142,Z 301.58,A -85,B 0,C 180,E1 -12434.596,E2 -12434.596} C_VEL
LIN {X 0,Y 378.763,Z 291.247,A -85,B 0,C 180,E1 -12435.608,E2 -12435.608} C_VEL
LIN {X 0,Y 379.469,Z 279.237,A -85,B 0,C 180,E1 -12436.544,E2 -12436.544} C_VEL
LIN {X 0,Y 379.898,Z 270.801,A -85,B 0,C 180,E1 -12437.079,E2 -12437.079} C_VEL
LIN {X 0,Y 377.515,Z 257.003,A -85,B 0,C 180,E1 -12437.842,E2 -12437.842} C_VEL
LIN {X 0,Y 375.907,Z 247.998,A -85,B 0,C 180,E1 -12438.248,E2 -12438.248} C_VEL
LIN {X 0,Y 376.21,Z 238.821,A -85,B 0,C 180,E1 -12441.939,E2 -12441.939} C_VEL
LIN {X 0,Y 376.437,Z 231.664,A -85,B 0,C 180,E1 -12444.839,E2 -12444.839} C_VEL
LIN {X 0,Y 376.708,Z 223.236,A -85,B 0,C 180,E1 -12448.275,E2 -12448.275} C_VEL
LIN {X 0,Y 377.091,Z 213.93,A -85,B 0,C 180,E1 -12452.085,E2 -12452.085} C_VEL
LIN {X 0,Y 377.285,Z 206.12,A -85,B 0,C 180,E1 -12455.273,E2 -12455.273} C_VEL
LIN {X 0,Y 376.802,Z 201.274,A -85,B 0,C 180,E1 -12457.313,E2 -12457.313} C_VEL
LIN {X 0,Y 376.014,Z 196.648,A -85,B 0,C 180,E1 -12459.383,E2 -12459.383} C_VEL
LIN {X 0,Y 375.939,Z 196.657,A -85,B 0,C 180,E1 -12463.189,E2 -12463.189} C_VEL
LIN {X 0,Y 375.94,Z 196.656,A -85,B 0,C 180,E1 -12466.81,E2 -12466.81} C_VEL
LIN {X 0,Y 375.952,Z 196.658,A -85,B 0,C 180,E1 -12470.535,E2 -12470.535} C_VEL
LIN {X 0,Y 375.962,Z 196.658,A -85,B 0,C 180,E1 -12473.496,E2 -12473.496} C_VEL
LIN {X 0,Y 375.962,Z 196.657,A -85,B 0,C 180,E1 -12475.887,E2 -12475.887} C_VEL
LIN {X 0,Y 375.879,Z 196.667,A -85,B 0,C 180,E1 -12479.327,E2 -12479.327} C_VEL
LIN {X 0,Y 375.896,Z 196.665,A -85,B 0,C 180,E1 -12479.68,E2 -12479.68} C_VEL
LIN {X 0,Y 375.895,Z 198.211,A -85,B 0,C 180,E1 -12481.492,E2 -12481.492} C_VEL
LIN {X 0,Y 375.839,Z 201.765,A -85,B 0,C 180,E1 -12484.526,E2 -12484.526} C_VEL
LIN {X 0,Y 375.784,Z 204.542,A -85,B 0,C 180,E1 -12486.873,E2 -12486.873} C_VEL
LIN {X 0,Y 375.679,Z 208.813,A -85,B 0,C 180,E1 -12490.321,E2 -12490.321} C_VEL
LIN {X 0,Y 375.695,Z 211.738,A -85,B 0,C 180,E1 -12492.583,E2 -12492.583} C_VEL
LIN {X 0,Y 375.711,Z 217.277,A -85,B 0,C 180,E1 -12496.584,E2 -12496.584} C_VEL
LIN {X 0,Y 375.768,Z 218.705,A -85,B 0,C 180,E1 -12497.424,E2 -12497.424} C_VEL
LIN {X 0,Y 378.067,Z 228.16,A -85,B 0,C 180,E1 -12497.927,E2 -12497.927} C_VEL
LIN {X 0,Y 379.643,Z 236.474,A -85,B 0,C 180,E1 -12498.52,E2 -12498.52} C_VEL
LIN {X 0,Y 379.36,Z 245.803,A -85,B 0,C 180,E1 -12499.322,E2 -12499.322} C_VEL
LIN {X 0,Y 378.921,Z 253.079,A -85,B 0,C 180,E1 -12500.15,E2 -12500.15} C_VEL
LIN {X 0,Y 378.508,Z 258.522,A -85,B 0,C 180,E1 -12500.918,E2 -12500.918} C_VEL
LIN {X 0,Y 377.988,Z 264.617,A -85,B 0,C 180,E1 -12501.983,E2 -12501.983} C_VEL
LIN {X 0,Y 377.425,Z 270.37,A -85,B 0,C 180,E1 -12503.315,E2 -12503.315} C_VEL
LIN {X 0,Y 377.087,Z 274.599,A -85,B 0,C 180,E1 -12504.652,E2 -12504.652} C_VEL
LIN {X 0,Y 376.797,Z 277.144,A -85,B 0,C 180,E1 -12505.72,E2 -12505.72} C_VEL
LIN {X 0,Y 376.389,Z 279.055,A -85,B 0,C 180,E1 -12506.787,E2 -12506.787} C_VEL
LIN {X 0,Y 376.32,Z 280.342,A -85,B 0,C 180,E1 -12507.858,E2 -12507.858} C_VEL
LIN {X 0,Y 376.182,Z 281.116,A -85,B 0,C 180,E1 -12508.928,E2 -12508.928} C_VEL
LIN {X 0,Y 376.124,Z 281.381,A -85,B 0,C 180,E1 -12509.999,E2 -12509.999} C_VEL
LIN {X 0,Y 376.177,Z 281.156,A -85,B 0,C 180,E1 -12511.069,E2 -12511.069} C_VEL
LIN {X 0,Y 376.309,Z 280.436,A -85,B 0,C 180,E1 -12512.139,E2 -12512.139} C_VEL
LIN {X 0,Y 376.385,Z 279.205,A -85,B 0,C 180,E1 -12513.21,E2 -12513.21} C_VEL
LIN {X 0,Y 376.996,Z 276.193,A -85,B 0,C 180,E1 -12514.811,E2 -12514.811} C_VEL
LIN {X 0,Y 377.178,Z 271.691,A -85,B 0,C 180,E1 -12516.418,E2 -12516.418} C_VEL
LIN {X 0,Y 377.646,Z 268.698,A -85,B 0,C 180,E1 -12517.215,E2 -12517.215} C_VEL
LIN {X 0,Y 377.943,Z 265.073,A -85,B 0,C 180,E1 -12518.015,E2 -12518.015} C_VEL
LIN {X 0,Y 378.498,Z 259.163,A -85,B 0,C 180,E1 -12519.079,E2 -12519.079} C_VEL
LIN {X 0,Y 379.013,Z 252.44,A -85,B 0,C 180,E1 -12520.034,E2 -12520.034} C_VEL
LIN {X 0,Y 379.419,Z 243.905,A -85,B 0,C 180,E1 -12520.97,E2 -12520.97} C_VEL
LIN {X 0,Y 379.673,Z 236.044,A -85,B 0,C 180,E1 -12521.612,E2 -12521.612} C_VEL
LIN {X 0,Y 377.651,Z 226.295,A -85,B 0,C 180,E1 -12522.288,E2 -12522.288} C_VEL
LIN {X 0,Y 375.726,Z 218.493,A -85,B 0,C 180,E1 -12522.695,E2 -12522.695} C_VEL
LIN {X 0,Y 375.644,Z 213.392,A -85,B 0,C 180,E1 -12526.297,E2 -12526.297} C_VEL
LIN {X 0,Y 375.659,Z 210.002,A -85,B 0,C 180,E1 -12528.863,E2 -12528.863} C_VEL
LIN {X 0,Y 374.987,Z 208.992,A -85,B 0,C 180,E1 -12529.744,E2 -12529.744} C_VEL
LIN {X 0,Y 372.148,Z 207.618,A -85,B 0,C 180,E1 -12531.186,E2 -12531.186} C_VEL
LIN {X 0,Y 369.789,Z 206.577,A -85,B 0,C 180,E1 -12532.353,E2 -12532.353} C_VEL
LIN {X 0,Y 368.831,Z 205.662,A -85,B 0,C 180,E1 -12533.252,E2 -12533.252} C_VEL
LIN {X 0,Y 368.782,Z 205.316,A -85,B 0,C 180,E1 -12533.555,E2 -12533.555} C_VEL
LIN {X 0,Y 368.848,Z 201.003,A -85,B 0,C 180,E1 -12537.211,E2 -12537.211} C_VEL
LIN {X 0,Y 368.842,Z 197.542,A -85,B 0,C 180,E1 -12540.325,E2 -12540.325} C_VEL
LIN {X 0,Y 368.891,Z 197.537,A -85,B 0,C 180,E1 -12543.537,E2 -12543.537} C_VEL
LIN {X 0,Y 368.898,Z 197.533,A -85,B 0,C 180,E1 -12546.855,E2 -12546.855} C_VEL
LIN {X 0,Y 368.906,Z 197.532,A -85,B 0,C 180,E1 -12550.369,E2 -12550.369} C_VEL
LIN {X 0,Y 368.877,Z 197.533,A -85,B 0,C 180,E1 -12553.615,E2 -12553.615} C_VEL
LIN {X 0,Y 368.878,Z 197.534,A -85,B 0,C 180,E1 -12556.694,E2 -12556.694} C_VEL
LIN {X 0,Y 368.905,Z 197.528,A -85,B 0,C 180,E1 -12559.641,E2 -12559.641} C_VEL
LIN {X 0,Y 368.895,Z 197.532,A -85,B 0,C 180,E1 -12563.143,E2 -12563.143} C_VEL
LIN {X 0,Y 368.892,Z 197.53,A -85,B 0,C 180,E1 -12566.461,E2 -12566.461} C_VEL
LIN {X 0,Y 368.915,Z 197.526,A -85,B 0,C 180,E1 -12570.309,E2 -12570.309} C_VEL
LIN {X 0,Y 368.972,Z 197.523,A -85,B 0,C 180,E1 -12573.534,E2 -12573.534} C_VEL
LIN {X 0,Y 368.956,Z 197.527,A -85,B 0,C 180,E1 -12576.421,E2 -12576.421} C_VEL
LIN {X 0,Y 368.926,Z 197.523,A -85,B 0,C 180,E1 -12579.946,E2 -12579.946} C_VEL
LIN {X 0,Y 368.968,Z 197.525,A -85,B 0,C 180,E1 -12583.398,E2 -12583.398} C_VEL
LIN {X 0,Y 369.047,Z 197.512,A -85,B 0,C 180,E1 -12586.79,E2 -12586.79} C_VEL
LIN {X 0,Y 369.057,Z 197.503,A -85,B 0,C 180,E1 -12590.131,E2 -12590.131} C_VEL
LIN {X 0,Y 369.187,Z 197.495,A -85,B 0,C 180,E1 -12593.441,E2 -12593.441} C_VEL
LIN {X 0,Y 369.307,Z 197.48,A -85,B 0,C 180,E1 -12597.819,E2 -12597.819} C_VEL
LIN {X 0,Y 369.446,Z 197.453,A -85,B 0,C 180,E1 -12600,E2 -12600} C_VEL
LIN {X 0,Y 369.303,Z 197.48,A -85,B 0,C 180,E1 -12602.181,E2 -12602.181} C_VEL
LIN {X 0,Y 369.194,Z 197.496,A -85,B 0,C 180,E1 -12606.558,E2 -12606.558} C_VEL
LIN {X 0,Y 369.126,Z 197.499,A -85,B 0,C 180,E1 -12608.761,E2 -12608.761} C_VEL
LIN {X 0,Y 368.993,Z 197.523,A -85,B 0,C 180,E1 -12612.094,E2 -12612.094} C_VEL
LIN {X 0,Y 368.985,Z 197.522,A -85,B 0,C 180,E1 -12615.465,E2 -12615.465} C_VEL
LIN {X 0,Y 368.942,Z 197.527,A -85,B 0,C 180,E1 -12618.895,E2 -12618.895} C_VEL
LIN {X 0,Y 368.908,Z 197.534,A -85,B 0,C 180,E1 -12622.397,E2 -12622.397} C_VEL
LIN {X 0,Y 368.908,Z 197.535,A -85,B 0,C 180,E1 -12625.987,E2 -12625.987} C_VEL
LIN {X 0,Y 368.882,Z 197.538,A -85,B 0,C 180,E1 -12629.693,E2 -12629.693} C_VEL
LIN {X 0,Y 368.887,Z 197.535,A -85,B 0,C 180,E1 -12633.044,E2 -12633.044} C_VEL
LIN {X 0,Y 368.907,Z 197.533,A -85,B 0,C 180,E1 -12636.198,E2 -12636.198} C_VEL
LIN {X 0,Y 368.866,Z 197.54,A -85,B 0,C 180,E1 -12638.958,E2 -12638.958} C_VEL
LIN {X 0,Y 368.863,Z 197.536,A -85,B 0,C 180,E1 -12642.009,E2 -12642.009} C_VEL
LIN {X 0,Y 368.872,Z 197.536,A -85,B 0,C 180,E1 -12645.177,E2 -12645.177} C_VEL
LIN {X 0,Y 368.911,Z 197.644,A -85,B 0,C 180,E1 -12648.472,E2 -12648.472} C_VEL
LIN {X 0,Y 371.094,Z 206.642,A -85,B 0,C 180,E1 -12651.665,E2 -12651.665} C_VEL
LIN {X 0,Y 373.709,Z 217.953,A -85,B 0,C 180,E1 -12655.33,E2 -12655.33} C_VEL
LIN {X 0,Y 375.503,Z 226.76,A -85,B 0,C 180,E1 -12657.937,E2 -12657.937} C_VEL
LIN {X 0,Y 375.445,Z 229.592,A -85,B 0,C 180,E1 -12658.706,E2 -12658.706} C_VEL
LIN {X 0,Y 373.009,Z 245.175,A -85,B 0,C 180,E1 -12662.674,E2 -12662.674} C_VEL
LIN {X 0,Y 371.063,Z 260.628,A -85,B 0,C 180,E1 -12666.565,E2 -12666.565} C_VEL
LIN {X 0,Y 369.508,Z 276.178,A -85,B 0,C 180,E1 -12670.56,E2 -12670.56} C_VEL
LIN {X 0,Y 369.183,Z 279.7,A -85,B 0,C 180,E1 -12671.486,E2 -12671.486} C_VEL
LIN {X 0,Y 370.922,Z 299.473,A -85,B 0,C 180,E1 -12672.196,E2 -12672.196} C_VEL
LIN {X 0,Y 371.655,Z 311.654,A -85,B 0,C 180,E1 -12672.816,E2 -12672.816} C_VEL
LIN {X 0,Y 371.632,Z 320.483,A -85,B 0,C 180,E1 -12673.381,E2 -12673.381} C_VEL
LIN {X 0,Y 370.912,Z 331.074,A -85,B 0,C 180,E1 -12674.196,E2 -12674.196} C_VEL
LIN {X 0,Y 370.227,Z 342.366,A -85,B 0,C 180,E1 -12675.293,E2 -12675.293} C_VEL
LIN {X 0,Y 369.434,Z 352.836,A -85,B 0,C 180,E1 -12676.555,E2 -12676.555} C_VEL
LIN {X 0,Y 368.831,Z 361.991,A -85,B 0,C 180,E1 -12677.902,E2 -12677.902} C_VEL
LIN {X 0,Y 368.19,Z 371.033,A -85,B 0,C 180,E1 -12679.554,E2 -12679.554} C_VEL
LIN {X 0,Y 367.887,Z 378.333,A -85,B 0,C 180,E1 -12681.211,E2 -12681.211} C_VEL
LIN {X 0,Y 367.732,Z 384.132,A -85,B 0,C 180,E1 -12682.865,E2 -12682.865} C_VEL
LIN {X 0,Y 367.663,Z 388.626,A -85,B 0,C 180,E1 -12684.517,E2 -12684.517} C_VEL
LIN {X 0,Y 367.646,Z 390.965,A -85,B 0,C 180,E1 -12685.616,E2 -12685.616} C_VEL
LIN {X 0,Y 367.673,Z 392.852,A -85,B 0,C 180,E1 -12686.714,E2 -12686.714} C_VEL
LIN {X 0,Y 367.741,Z 394.252,A -85,B 0,C 180,E1 -12687.811,E2 -12687.811} C_VEL
LIN {X 0,Y 367.728,Z 395.192,A -85,B 0,C 180,E1 -12688.906,E2 -12688.906} C_VEL
LIN {X 0,Y 367.754,Z 395.716,A -85,B 0,C 180,E1 -12690.001,E2 -12690.001} C_VEL
LIN {X 0,Y 367.709,Z 395.801,A -85,B 0,C 180,E1 -12691.097,E2 -12691.097} C_VEL
LIN {X 0,Y 367.704,Z 395.424,A -85,B 0,C 180,E1 -12692.192,E2 -12692.192} C_VEL
LIN {X 0,Y 367.584,Z 394.626,A -85,B 0,C 180,E1 -12693.29,E2 -12693.29} C_VEL
LIN {X 0,Y 367.61,Z 393.423,A -85,B 0,C 180,E1 -12694.387,E2 -12694.387} C_VEL
LIN {X 0,Y 367.586,Z 390.514,A -85,B 0,C 180,E1 -12696.169,E2 -12696.169} C_VEL
LIN {X 0,Y 367.859,Z 385.594,A -85,B 0,C 180,E1 -12698.24,E2 -12698.24} C_VEL
LIN {X 0,Y 368.254,Z 380.43,A -85,B 0,C 180,E1 -12699.892,E2 -12699.892} C_VEL
LIN {X 0,Y 368.855,Z 374.001,A -85,B 0,C 180,E1 -12701.542,E2 -12701.542} C_VEL
LIN {X 0,Y 369.91,Z 366.123,A -85,B 0,C 180,E1 -12703.18,E2 -12703.18} C_VEL
LIN {X 0,Y 370.92,Z 356.286,A -85,B 0,C 180,E1 -12704.853,E2 -12704.853} C_VEL
LIN {X 0,Y 372.3,Z 346.743,A -85,B 0,C 180,E1 -12706.168,E2 -12706.168} C_VEL
LIN {X 0,Y 373.88,Z 334.818,A -85,B 0,C 180,E1 -12707.504,E2 -12707.504} C_VEL
LIN {X 0,Y 375.392,Z 323.114,A -85,B 0,C 180,E1 -12708.56,E2 -12708.56} C_VEL
LIN {X 0,Y 376.015,Z 308.516,A -85,B 0,C 180,E1 -12709.661,E2 -12709.661} C_VEL
LIN {X 0,Y 375.299,Z 294.609,A -85,B 0,C 180,E1 -12710.557,E2 -12710.557} C_VEL
LIN {X 0,Y 373.218,Z 280.677,A -85,B 0,C 180,E1 -12711.39,E2 -12711.39} C_VEL
LIN {X 0,Y 372.075,Z 274.665,A -85,B 0,C 180,E1 -12711.802,E2 -12711.802} C_VEL
LIN {X 0,Y 371.295,Z 262.858,A -85,B 0,C 180,E1 -12713.275,E2 -12713.275} C_VEL
LIN {X 0,Y 371.228,Z 259.143,A -85,B 0,C 180,E1 -12713.797,E2 -12713.797} C_VEL
LIN {X 0,Y 373.249,Z 243.457,A -85,B 0,C 180,E1 -12717.751,E2 -12717.751} C_VEL
LIN {X 0,Y 375.572,Z 228.313,A -85,B 0,C 180,E1 -12721.599,E2 -12721.599} C_VEL
LIN {X 0,Y 374.879,Z 223.674,A -85,B 0,C 180,E1 -12722.935,E2 -12722.935} C_VEL
LIN {X 0,Y 372.786,Z 214.112,A -85,B 0,C 180,E1 -12725.839,E2 -12725.839} C_VEL
LIN {X 0,Y 371.971,Z 210.612,A -85,B 0,C 180,E1 -12727.032,E2 -12727.032} C_VEL
LIN {X 0,Y 372.878,Z 208.582,A -85,B 0,C 180,E1 -12729.397,E2 -12729.397} C_VEL
LIN {X 0,Y 372.953,Z 208.486,A -85,B 0,C 180,E1 -12731.267,E2 -12731.267} C_VEL
LIN {X 0,Y 373.212,Z 209.826,A -85,B 0,C 180,E1 -12734.309,E2 -12734.309} C_VEL
LIN {X 0,Y 373.758,Z 212.602,A -85,B 0,C 180,E1 -12737.396,E2 -12737.396} C_VEL
LIN {X 0,Y 374.409,Z 216.306,A -85,B 0,C 180,E1 -12740.341,E2 -12740.341} C_VEL
LIN {X 0,Y 374.918,Z 220.598,A -85,B 0,C 180,E1 -12743.14,E2 -12743.14} C_VEL
LIN {X 0,Y 374.927,Z 223.1,A -85,B 0,C 180,E1 -12744.472,E2 -12744.472} C_VEL
LIN {X 0,Y 373.404,Z 232.258,A -85,B 0,C 180,E1 -12748.829,E2 -12748.829} C_VEL
LIN {X 0,Y 372.514,Z 240.144,A -85,B 0,C 180,E1 -12752.466,E2 -12752.466} C_VEL
LIN {X 0,Y 371.813,Z 248.033,A -85,B 0,C 180,E1 -12756.022,E2 -12756.022} C_VEL
LIN {X 0,Y 371.396,Z 253.416,A -85,B 0,C 180,E1 -12758.345,E2 -12758.345} C_VEL
LIN {X 0,Y 375.465,Z 264.896,A -85,B 0,C 180,E1 -12759.377,E2 -12759.377} C_VEL
LIN {X 0,Y 377.989,Z 274.997,A -85,B 0,C 180,E1 -12760.291,E2 -12760.291} C_VEL
LIN {X 0,Y 378.507,Z 278.67,A -85,B 0,C 180,E1 -12760.617,E2 -12760.617} C_VEL
LIN {X 0,Y 377.232,Z 290.523,A -85,B 0,C 180,E1 -12761.535,E2 -12761.535} C_VEL
LIN {X 0,Y 375.677,Z 302.986,A -85,B 0,C 180,E1 -12762.77,E2 -12762.77} C_VEL
LIN {X 0,Y 374.41,Z 312.456,A -85,B 0,C 180,E1 -12763.926,E2 -12763.926} C_VEL
LIN {X 0,Y 372.773,Z 323.152,A -85,B 0,C 180,E1 -12765.534,E2 -12765.534} C_VEL
LIN {X 0,Y 371.41,Z 331.795,A -85,B 0,C 180,E1 -12767.154,E2 -12767.154} C_VEL
LIN {X 0,Y 370.368,Z 339.797,A -85,B 0,C 180,E1 -12769.061,E2 -12769.061} C_VEL
LIN {X 0,Y 369.484,Z 345.252,A -85,B 0,C 180,E1 -12770.696,E2 -12770.696} C_VEL
LIN {X 0,Y 368.865,Z 349.527,A -85,B 0,C 180,E1 -12772.336,E2 -12772.336} C_VEL
LIN {X 0,Y 368.377,Z 351.772,A -85,B 0,C 180,E1 -12773.427,E2 -12773.427} C_VEL
LIN {X 0,Y 368.297,Z 353.559,A -85,B 0,C 180,E1 -12774.525,E2 -12774.525} C_VEL
LIN {X 0,Y 368.169,Z 354.953,A -85,B 0,C 180,E1 -12775.621,E2 -12775.621} C_VEL
LIN {X 0,Y 367.944,Z 355.902,A -85,B 0,C 180,E1 -12776.715,E2 -12776.715} C_VEL
LIN {X 0,Y 367.764,Z 356.45,A -85,B 0,C 180,E1 -12777.81,E2 -12777.81} C_VEL
LIN {X 0,Y 367.642,Z 356.605,A -85,B 0,C 180,E1 -12778.905,E2 -12778.905} C_VEL
LIN {X 0,Y 367.586,Z 356.328,A -85,B 0,C 180,E1 -12780,E2 -12780} C_VEL
LIN {X 0,Y 367.608,Z 355.618,A -85,B 0,C 180,E1 -12781.096,E2 -12781.096} C_VEL
LIN {X 0,Y 367.666,Z 354.511,A -85,B 0,C 180,E1 -12782.191,E2 -12782.191} C_VEL
LIN {X 0,Y 367.687,Z 352.04,A -85,B 0,C 180,E1 -12783.836,E2 -12783.836} C_VEL
LIN {X 0,Y 367.86,Z 348.55,A -85,B 0,C 180,E1 -12785.482,E2 -12785.482} C_VEL
LIN {X 0,Y 368.081,Z 343.878,A -85,B 0,C 180,E1 -12787.149,E2 -12787.149} C_VEL
LIN {X 0,Y 368.52,Z 336.998,A -85,B 0,C 180,E1 -12789.052,E2 -12789.052} C_VEL
LIN {X 0,Y 369.07,Z 329.47,A -85,B 0,C 180,E1 -12790.7,E2 -12790.7} C_VEL
LIN {X 0,Y 369.59,Z 321.831,A -85,B 0,C 180,E1 -12792.074,E2 -12792.074} C_VEL
LIN {X 0,Y 370.466,Z 311.585,A -85,B 0,C 180,E1 -12793.578,E2 -12793.578} C_VEL
LIN {X 0,Y 371.238,Z 300.318,A -85,B 0,C 180,E1 -12794.923,E2 -12794.923} C_VEL
LIN {X 0,Y 371.957,Z 288.517,A -85,B 0,C 180,E1 -12796.042,E2 -12796.042} C_VEL
LIN {X 0,Y 372.764,Z 275.774,A -85,B 0,C 180,E1 -12796.992,E2 -12796.992} C_VEL
LIN {X 0,Y 372.831,Z 271.335,A -85,B 0,C 180,E1 -12797.271,E2 -12797.271} C_VEL
LIN {X 0,Y 370.517,Z 257.442,A -85,B 0,C 180,E1 -12798.055,E2 -12798.055} C_VEL
LIN {X 0,Y 368.854,Z 248.363,A -85,B 0,C 180,E1 -12798.461,E2 -12798.461} C_VEL
LIN {X 0,Y 369.217,Z 238.714,A -85,B 0,C 180,E1 -12802.377,E2 -12802.377} C_VEL
LIN {X 0,Y 369.439,Z 231.461,A -85,B 0,C 180,E1 -12805.343,E2 -12805.343} C_VEL
LIN {X 0,Y 369.75,Z 222.498,A -85,B 0,C 180,E1 -12809.031,E2 -12809.031} C_VEL
LIN {X 0,Y 370.088,Z 215.021,A -85,B 0,C 180,E1 -12812.122,E2 -12812.122} C_VEL
LIN {X 0,Y 370.288,Z 207.339,A -85,B 0,C 180,E1 -12815.299,E2 -12815.299} C_VEL
LIN {X 0,Y 369.793,Z 202.296,A -85,B 0,C 180,E1 -12817.457,E2 -12817.457} C_VEL
LIN {X 0,Y 368.971,Z 197.526,A -85,B 0,C 180,E1 -12819.562,E2 -12819.562} C_VEL
LIN {X 0,Y 368.888,Z 197.535,A -85,B 0,C 180,E1 -12823.615,E2 -12823.615} C_VEL
LIN {X 0,Y 368.891,Z 197.534,A -85,B 0,C 180,E1 -12826.695,E2 -12826.695} C_VEL
LIN {X 0,Y 368.914,Z 197.533,A -85,B 0,C 180,E1 -12829.643,E2 -12829.643} C_VEL
LIN {X 0,Y 368.901,Z 197.536,A -85,B 0,C 180,E1 -12833.145,E2 -12833.145} C_VEL
LIN {X 0,Y 368.899,Z 197.536,A -85,B 0,C 180,E1 -12836.461,E2 -12836.461} C_VEL
LIN {X 0,Y 368.859,Z 197.541,A -85,B 0,C 180,E1 -12839.039,E2 -12839.039} C_VEL
LIN {X 0,Y 368.84,Z 198.02,A -85,B 0,C 180,E1 -12840.302,E2 -12840.302} C_VEL
LIN {X 0,Y 368.853,Z 201.751,A -85,B 0,C 180,E1 -12843.576,E2 -12843.576} C_VEL
LIN {X 0,Y 368.803,Z 205.11,A -85,B 0,C 180,E1 -12846.409,E2 -12846.409} C_VEL
LIN {X 0,Y 368.647,Z 209.403,A -85,B 0,C 180,E1 -12849.929,E2 -12849.929} C_VEL
LIN {X 0,Y 368.695,Z 212.545,A -85,B 0,C 180,E1 -12852.382,E2 -12852.382} C_VEL
LIN {X 0,Y 368.696,Z 218.624,A -85,B 0,C 180,E1 -12856.776,E2 -12856.776} C_VEL
LIN {X 0,Y 368.715,Z 219.085,A -85,B 0,C 180,E1 -12857.092,E2 -12857.092} C_VEL
LIN {X 0,Y 371.555,Z 230.933,A -85,B 0,C 180,E1 -12857.782,E2 -12857.782} C_VEL
LIN {X 0,Y 372.787,Z 237.864,A -85,B 0,C 180,E1 -12858.306,E2 -12858.306} C_VEL
LIN {X 0,Y 372.495,Z 246.99,A -85,B 0,C 180,E1 -12859.123,E2 -12859.123} C_VEL
LIN {X 0,Y 372.024,Z 254.142,A -85,B 0,C 180,E1 -12859.957,E2 -12859.957} C_VEL
LIN {X 0,Y 371.585,Z 259.594,A -85,B 0,C 180,E1 -12860.747,E2 -12860.747} C_VEL
LIN {X 0,Y 371.033,Z 265.65,A -85,B 0,C 180,E1 -12861.831,E2 -12861.831} C_VEL
LIN {X 0,Y 370.606,Z 270.341,A -85,B 0,C 180,E1 -12862.918,E2 -12862.918} C_VEL
LIN {X 0,Y 370.128,Z 274.066,A -85,B 0,C 180,E1 -12864.004,E2 -12864.004} C_VEL
LIN {X 0,Y 370.006,Z 276.935,A -85,B 0,C 180,E1 -12865.095,E2 -12865.095} C_VEL
LIN {X 0,Y 369.375,Z 280.032,A -85,B 0,C 180,E1 -12866.726,E2 -12866.726} C_VEL
LIN {X 0,Y 369.3,Z 281.317,A -85,B 0,C 180,E1 -12867.817,E2 -12867.817} C_VEL
LIN {X 0,Y 369.157,Z 282.09,A -85,B 0,C 180,E1 -12868.908,E2 -12868.908} C_VEL
LIN {X 0,Y 369.098,Z 282.355,A -85,B 0,C 180,E1 -12869.999,E2 -12869.999} C_VEL
LIN {X 0,Y 369.153,Z 282.129,A -85,B 0,C 180,E1 -12871.089,E2 -12871.089} C_VEL
LIN {X 0,Y 369.29,Z 281.41,A -85,B 0,C 180,E1 -12872.18,E2 -12872.18} C_VEL
LIN {X 0,Y 369.371,Z 280.181,A -85,B 0,C 180,E1 -12873.271,E2 -12873.271} C_VEL
LIN {X 0,Y 369.998,Z 277.178,A -85,B 0,C 180,E1 -12874.902,E2 -12874.902} C_VEL
LIN {X 0,Y 370.195,Z 272.692,A -85,B 0,C 180,E1 -12876.539,E2 -12876.539} C_VEL
LIN {X 0,Y 370.677,Z 269.708,A -85,B 0,C 180,E1 -12877.351,E2 -12877.351} C_VEL
LIN {X 0,Y 370.988,Z 266.11,A -85,B 0,C 180,E1 -12878.167,E2 -12878.167} C_VEL
LIN {X 0,Y 371.576,Z 260.23,A -85,B 0,C 180,E1 -12879.25,E2 -12879.25} C_VEL
LIN {X 0,Y 372.118,Z 253.49,A -85,B 0,C 180,E1 -12880.23,E2 -12880.23} C_VEL
LIN {X 0,Y 372.564,Z 244.779,A -85,B 0,C 180,E1 -12881.209,E2 -12881.209} C_VEL
LIN {X 0,Y 372.85,Z 237.416,A -85,B 0,C 180,E1 -12881.827,E2 -12881.827} C_VEL
LIN {X 0,Y 370.902,Z 227.986,A -85,B 0,C 180,E1 -12882.515,E2 -12882.515} C_VEL
LIN {X 0,Y 368.703,Z 219.096,A -85,B 0,C 180,E1 -12883.011,E2 -12883.011} C_VEL
LIN {X 0,Y 368.623,Z 214.049,A -85,B 0,C 180,E1 -12886.616,E2 -12886.616} C_VEL
LIN {X 0,Y 368.641,Z 211.023,A -85,B 0,C 180,E1 -12888.909,E2 -12888.909} C_VEL
LIN {X 0,Y 368.728,Z 206.671,A -85,B 0,C 180,E1 -12892.406,E2 -12892.406} C_VEL
LIN {X 0,Y 368.782,Z 205.316,A -85,B 0,C 180,E1 -12893.555,E2 -12893.555} C_VEL
LIN {X 0,Y 368.196,Z 204.37,A -85,B 0,C 180,E1 -12894.455,E2 -12894.455} C_VEL
LIN {X 0,Y 365.389,Z 203.066,A -85,B 0,C 180,E1 -12895.927,E2 -12895.927} C_VEL
LIN {X 0,Y 362.964,Z 202.068,A -85,B 0,C 180,E1 -12897.118,E2 -12897.118} C_VEL
LIN {X 0,Y 361.915,Z 201.168,A -85,B 0,C 180,E1 -12898.037,E2 -12898.037} C_VEL
LIN {X 0,Y 361.829,Z 200.824,A -85,B 0,C 180,E1 -12898.346,E2 -12898.346} C_VEL
LIN {X 0,Y 361.819,Z 198.585,A -85,B 0,C 180,E1 -12900.331,E2 -12900.331} C_VEL
LIN {X 0,Y 361.853,Z 198.413,A -85,B 0,C 180,E1 -12903.367,E2 -12903.367} C_VEL
LIN {X 0,Y 361.868,Z 198.41,A -85,B 0,C 180,E1 -12907.016,E2 -12907.016} C_VEL
LIN {X 0,Y 361.85,Z 198.411,A -85,B 0,C 180,E1 -12909.86,E2 -12909.86} C_VEL
LIN {X 0,Y 361.83,Z 198.415,A -85,B 0,C 180,E1 -12912.827,E2 -12912.827} C_VEL
LIN {X 0,Y 361.821,Z 198.413,A -85,B 0,C 180,E1 -12915.943,E2 -12915.943} C_VEL
LIN {X 0,Y 361.829,Z 198.41,A -85,B 0,C 180,E1 -12919.243,E2 -12919.243} C_VEL
LIN {X 0,Y 361.857,Z 198.407,A -85,B 0,C 180,E1 -12922.775,E2 -12922.775} C_VEL
LIN {X 0,Y 361.848,Z 198.408,A -85,B 0,C 180,E1 -12925.719,E2 -12925.719} C_VEL
LIN {X 0,Y 361.867,Z 198.406,A -85,B 0,C 180,E1 -12929.671,E2 -12929.671} C_VEL
LIN {X 0,Y 361.945,Z 198.398,A -85,B 0,C 180,E1 -12933.474,E2 -12933.474} C_VEL
LIN {X 0,Y 361.88,Z 198.406,A -85,B 0,C 180,E1 -12937.144,E2 -12937.144} C_VEL
LIN {X 0,Y 361.91,Z 198.399,A -85,B 0,C 180,E1 -12940.723,E2 -12940.723} C_VEL
LIN {X 0,Y 361.938,Z 198.391,A -85,B 0,C 180,E1 -12944.226,E2 -12944.226} C_VEL
LIN {X 0,Y 361.988,Z 198.391,A -85,B 0,C 180,E1 -12946.527,E2 -12946.527} C_VEL
LIN {X 0,Y 362.021,Z 198.38,A -85,B 0,C 180,E1 -12949.938,E2 -12949.938} C_VEL
LIN {X 0,Y 362.149,Z 198.373,A -85,B 0,C 180,E1 -12953.313,E2 -12953.313} C_VEL
LIN {X 0,Y 362.271,Z 198.356,A -85,B 0,C 180,E1 -12957.776,E2 -12957.776} C_VEL
LIN {X 0,Y 362.416,Z 198.329,A -85,B 0,C 180,E1 -12960,E2 -12960} C_VEL
LIN {X 0,Y 362.267,Z 198.357,A -85,B 0,C 180,E1 -12962.224,E2 -12962.224} C_VEL
LIN {X 0,Y 362.158,Z 198.374,A -85,B 0,C 180,E1 -12966.686,E2 -12966.686} C_VEL
LIN {X 0,Y 362.062,Z 198.378,A -85,B 0,C 180,E1 -12968.933,E2 -12968.933} C_VEL
LIN {X 0,Y 361.948,Z 198.398,A -85,B 0,C 180,E1 -12972.333,E2 -12972.333} C_VEL
LIN {X 0,Y 361.95,Z 198.399,A -85,B 0,C 180,E1 -12974.621,E2 -12974.621} C_VEL
LIN {X 0,Y 361.9,Z 198.401,A -85,B 0,C 180,E1 -12978.102,E2 -12978.102} C_VEL
LIN {X 0,Y 361.849,Z 198.414,A -85,B 0,C 180,E1 -12981.656,E2 -12981.656} C_VEL
LIN {X 0,Y 361.855,Z 198.413,A -85,B 0,C 180,E1 -12985.296,E2 -12985.296} C_VEL
LIN {X 0,Y 361.845,Z 198.413,A -85,B 0,C 180,E1 -12989.075,E2 -12989.075} C_VEL
LIN {X 0,Y 361.839,Z 198.413,A -85,B 0,C 180,E1 -12992.946,E2 -12992.946} C_VEL
LIN {X 0,Y 361.858,Z 198.414,A -85,B 0,C 180,E1 -12995.638,E2 -12995.638} C_VEL
LIN {X 0,Y 361.817,Z 198.417,A -85,B 0,C 180,E1 -12999.019,E2 -12999.019} C_VEL
LIN {X 0,Y 361.825,Z 198.42,A -85,B 0,C 180,E1 -13002.831,E2 -13002.831} C_VEL
LIN {X 0,Y 361.811,Z 198.416,A -85,B 0,C 180,E1 -13005.948,E2 -13005.948} C_VEL
LIN {X 0,Y 361.859,Z 198.549,A -85,B 0,C 180,E1 -13007.883,E2 -13007.883} C_VEL
LIN {X 0,Y 363.707,Z 205.954,A -85,B 0,C 180,E1 -13010.618,E2 -13010.618} C_VEL
LIN {X 0,Y 366.244,Z 216.963,A -85,B 0,C 180,E1 -13014.347,E2 -13014.347} C_VEL
LIN {X 0,Y 368.291,Z 226.518,A -85,B 0,C 180,E1 -13017.304,E2 -13017.304} C_VEL
LIN {X 0,Y 368.631,Z 230.292,A -85,B 0,C 180,E1 -13018.381,E2 -13018.381} C_VEL
LIN {X 0,Y 366.21,Z 245.064,A -85,B 0,C 180,E1 -13022.245,E2 -13022.245} C_VEL
LIN {X 0,Y 364.225,Z 259.928,A -85,B 0,C 180,E1 -13026.097,E2 -13026.097} C_VEL
LIN {X 0,Y 362.547,Z 275.358,A -85,B 0,C 180,E1 -13030.171,E2 -13030.171} C_VEL
LIN {X 0,Y 362.192,Z 279.336,A -85,B 0,C 180,E1 -13031.242,E2 -13031.242} C_VEL
LIN {X 0,Y 363.852,Z 298.982,A -85,B 0,C 180,E1 -13031.969,E2 -13031.969} C_VEL
LIN {X 0,Y 364.648,Z 311.427,A -85,B 0,C 180,E1 -13032.62,E2 -13032.62} C_VEL
LIN {X 0,Y 364.651,Z 320.216,A -85,B 0,C 180,E1 -13033.198,E2 -13033.198} C_VEL
LIN {X 0,Y 363.813,Z 332.292,A -85,B 0,C 180,E1 -13034.167,E2 -13034.167} C_VEL
LIN {X 0,Y 362.94,Z 344.472,A -85,B 0,C 180,E1 -13035.422,E2 -13035.422} C_VEL
LIN {X 0,Y 362.188,Z 355.247,A -85,B 0,C 180,E1 -13036.822,E2 -13036.822} C_VEL
LIN {X 0,Y 361.602,Z 364.051,A -85,B 0,C 180,E1 -13038.226,E2 -13038.226} C_VEL
LIN {X 0,Y 361.04,Z 372.652,A -85,B 0,C 180,E1 -13039.912,E2 -13039.912} C_VEL
LIN {X 0,Y 360.766,Z 379.507,A -85,B 0,C 180,E1 -13041.6,E2 -13041.6} C_VEL
LIN {X 0,Y 360.601,Z 384.951,A -85,B 0,C 180,E1 -13043.286,E2 -13043.286} C_VEL
LIN {X 0,Y 360.628,Z 389.16,A -85,B 0,C 180,E1 -13044.97,E2 -13044.97} C_VEL
LIN {X 0,Y 360.584,Z 392.219,A -85,B 0,C 180,E1 -13046.649,E2 -13046.649} C_VEL
LIN {X 0,Y 360.674,Z 393.699,A -85,B 0,C 180,E1 -13047.768,E2 -13047.768} C_VEL
LIN {X 0,Y 360.656,Z 394.68,A -85,B 0,C 180,E1 -13048.885,E2 -13048.885} C_VEL
LIN {X 0,Y 360.679,Z 395.242,A -85,B 0,C 180,E1 -13050.001,E2 -13050.001} C_VEL
LIN {X 0,Y 360.638,Z 395.384,A -85,B 0,C 180,E1 -13051.118,E2 -13051.118} C_VEL
LIN {X 0,Y 360.602,Z 395.062,A -85,B 0,C 180,E1 -13052.235,E2 -13052.235} C_VEL
LIN {X 0,Y 360.531,Z 393.141,A -85,B 0,C 180,E1 -13054.474,E2 -13054.474} C_VEL
LIN {X 0,Y 360.5,Z 390.586,A -85,B 0,C 180,E1 -13056.144,E2 -13056.144} C_VEL
LIN {X 0,Y 360.693,Z 386.976,A -85,B 0,C 180,E1 -13057.841,E2 -13057.841} C_VEL
LIN {X 0,Y 361.054,Z 382.303,A -85,B 0,C 180,E1 -13059.525,E2 -13059.525} C_VEL
LIN {X 0,Y 361.75,Z 375.336,A -85,B 0,C 180,E1 -13061.488,E2 -13061.488} C_VEL
LIN {X 0,Y 363.008,Z 366.499,A -85,B 0,C 180,E1 -13063.435,E2 -13063.435} C_VEL
LIN {X 0,Y 364.047,Z 357.291,A -85,B 0,C 180,E1 -13065.073,E2 -13065.073} C_VEL
LIN {X 0,Y 365.712,Z 346.569,A -85,B 0,C 180,E1 -13066.611,E2 -13066.611} C_VEL
LIN {X 0,Y 367.405,Z 334.812,A -85,B 0,C 180,E1 -13067.967,E2 -13067.967} C_VEL
LIN {X 0,Y 368.991,Z 323.324,A -85,B 0,C 180,E1 -13069.038,E2 -13069.038} C_VEL
LIN {X 0,Y 369.676,Z 309.693,A -85,B 0,C 180,E1 -13070.119,E2 -13070.119} C_VEL
LIN {X 0,Y 369.106,Z 295.558,A -85,B 0,C 180,E1 -13071.094,E2 -13071.094} C_VEL
LIN {X 0,Y 367.264,Z 282.677,A -85,B 0,C 180,E1 -13071.919,E2 -13071.919} C_VEL
LIN {X 0,Y 365.749,Z 274.42,A -85,B 0,C 180,E1 -13072.493,E2 -13072.493} C_VEL
LIN {X 0,Y 365.146,Z 262.122,A -85,B 0,C 180,E1 -13074.143,E2 -13074.143} C_VEL
LIN {X 0,Y 364.932,Z 253.999,A -85,B 0,C 180,E1 -13075.427,E2 -13075.427} C_VEL
LIN {X 0,Y 367.243,Z 238.196,A -85,B 0,C 180,E1 -13079.525,E2 -13079.525} C_VEL
LIN {X 0,Y 368.609,Z 230.154,A -85,B 0,C 180,E1 -13081.624,E2 -13081.624} C_VEL
LIN {X 0,Y 368.133,Z 225.919,A -85,B 0,C 180,E1 -13082.86,E2 -13082.86} C_VEL
LIN {X 0,Y 366.183,Z 216.903,A -85,B 0,C 180,E1 -13085.665,E2 -13085.665} C_VEL
LIN {X 0,Y 366.692,Z 213.878,A -85,B 0,C 180,E1 -13088.205,E2 -13088.205} C_VEL
LIN {X 0,Y 367.091,Z 213.06,A -85,B 0,C 180,E1 -13089.184,E2 -13089.184} C_VEL
LIN {X 0,Y 367.202,Z 212.645,A -85,B 0,C 180,E1 -13090.599,E2 -13090.599} C_VEL
LIN {X 0,Y 367.209,Z 213.335,A -85,B 0,C 180,E1 -13093.553,E2 -13093.553} C_VEL
LIN {X 0,Y 367.506,Z 215.51,A -85,B 0,C 180,E1 -13096.611,E2 -13096.611} C_VEL
LIN {X 0,Y 367.985,Z 218.655,A -85,B 0,C 180,E1 -13099.507,E2 -13099.507} C_VEL
LIN {X 0,Y 368.361,Z 221.291,A -85,B 0,C 180,E1 -13101.468,E2 -13101.468} C_VEL
LIN {X 0,Y 368.552,Z 224.847,A -85,B 0,C 180,E1 -13103.762,E2 -13103.762} C_VEL
LIN {X 0,Y 368.004,Z 228.165,A -85,B 0,C 180,E1 -13105.468,E2 -13105.468} C_VEL
LIN {X 0,Y 366.54,Z 236.736,A -85,B 0,C 180,E1 -13109.637,E2 -13109.637} C_VEL
LIN {X 0,Y 365.641,Z 244.195,A -85,B 0,C 180,E1 -13113.148,E2 -13113.148} C_VEL
LIN {X 0,Y 364.883,Z 252.017,A -85,B 0,C 180,E1 -13116.743,E2 -13116.743} C_VEL
LIN {X 0,Y 364.734,Z 253.95,A -85,B 0,C 180,E1 -13117.599,E2 -13117.599} C_VEL
LIN {X 0,Y 369.287,Z 266.707,A -85,B 0,C 180,E1 -13118.835,E2 -13118.835} C_VEL
LIN {X 0,Y 371.812,Z 276.845,A -85,B 0,C 180,E1 -13119.82,E2 -13119.82} C_VEL
LIN {X 0,Y 372.284,Z 280.158,A -85,B 0,C 180,E1 -13120.135,E2 -13120.135} C_VEL
LIN {X 0,Y 370.955,Z 291.685,A -85,B 0,C 180,E1 -13121.068,E2 -13121.068} C_VEL
LIN {X 0,Y 369.334,Z 303.558,A -85,B 0,C 180,E1 -13122.274,E2 -13122.274} C_VEL
LIN {X 0,Y 367.782,Z 314.234,A -85,B 0,C 180,E1 -13123.629,E2 -13123.629} C_VEL
LIN {X 0,Y 366.043,Z 324.675,A -85,B 0,C 180,E1 -13125.262,E2 -13125.262} C_VEL
LIN {X 0,Y 364.621,Z 333.044,A -85,B 0,C 180,E1 -13126.91,E2 -13126.91} C_VEL
LIN {X 0,Y 363.648,Z 339.853,A -85,B 0,C 180,E1 -13128.574,E2 -13128.574} C_VEL
LIN {X 0,Y 362.547,Z 346.174,A -85,B 0,C 180,E1 -13130.516,E2 -13130.516} C_VEL
LIN {X 0,Y 361.862,Z 350.325,A -85,B 0,C 180,E1 -13132.186,E2 -13132.186} C_VEL
LIN {X 0,Y 361.367,Z 352.507,A -85,B 0,C 180,E1 -13133.299,E2 -13133.299} C_VEL
LIN {X 0,Y 361.26,Z 354.244,A -85,B 0,C 180,E1 -13134.418,E2 -13134.418} C_VEL
LIN {X 0,Y 361.132,Z 355.549,A -85,B 0,C 180,E1 -13135.535,E2 -13135.535} C_VEL
LIN {X 0,Y 360.898,Z 356.439,A -85,B 0,C 180,E1 -13136.651,E2 -13136.651} C_VEL
LIN {X 0,Y 360.706,Z 356.939,A -85,B 0,C 180,E1 -13137.767,E2 -13137.767} C_VEL
LIN {X 0,Y 360.577,Z 357.036,A -85,B 0,C 180,E1 -13138.883,E2 -13138.883} C_VEL
LIN {X 0,Y 360.52,Z 356.679,A -85,B 0,C 180,E1 -13140,E2 -13140} C_VEL
LIN {X 0,Y 360.544,Z 355.921,A -85,B 0,C 180,E1 -13141.117,E2 -13141.117} C_VEL
LIN {X 0,Y 360.573,Z 354.768,A -85,B 0,C 180,E1 -13142.234,E2 -13142.234} C_VEL
LIN {X 0,Y 360.605,Z 352.203,A -85,B 0,C 180,E1 -13143.911,E2 -13143.911} C_VEL
LIN {X 0,Y 360.788,Z 348.617,A -85,B 0,C 180,E1 -13145.589,E2 -13145.589} C_VEL
LIN {X 0,Y 361.019,Z 343.905,A -85,B 0,C 180,E1 -13147.27,E2 -13147.27} C_VEL
LIN {X 0,Y 361.473,Z 336.788,A -85,B 0,C 180,E1 -13149.23,E2 -13149.23} C_VEL
LIN {X 0,Y 362.05,Z 329.13,A -85,B 0,C 180,E1 -13150.91,E2 -13150.91} C_VEL
LIN {X 0,Y 362.783,Z 319.572,A -85,B 0,C 180,E1 -13152.588,E2 -13152.588} C_VEL
LIN {X 0,Y 363.504,Z 309.845,A -85,B 0,C 180,E1 -13153.986,E2 -13153.986} C_VEL
LIN {X 0,Y 364.258,Z 298.857,A -85,B 0,C 180,E1 -13155.266,E2 -13155.266} C_VEL
LIN {X 0,Y 365.064,Z 287.295,A -85,B 0,C 180,E1 -13156.353,E2 -13156.353} C_VEL
LIN {X 0,Y 365.877,Z 274.021,A -85,B 0,C 180,E1 -13157.322,E2 -13157.322} C_VEL
LIN {X 0,Y 365.145,Z 267.878,A -85,B 0,C 180,E1 -13157.719,E2 -13157.719} C_VEL
LIN {X 0,Y 362.807,Z 254.399,A -85,B 0,C 180,E1 -13158.441,E2 -13158.441} C_VEL
LIN {X 0,Y 361.837,Z 248.692,A -85,B 0,C 180,E1 -13158.692,E2 -13158.692} C_VEL
LIN {X 0,Y 362.153,Z 240.024,A -85,B 0,C 180,E1 -13162.236,E2 -13162.236} C_VEL
LIN {X 0,Y 362.395,Z 232.707,A -85,B 0,C 180,E1 -13165.255,E2 -13165.255} C_VEL
LIN {X 0,Y 362.729,Z 223.753,A -85,B 0,C 180,E1 -13168.972,E2 -13168.972} C_VEL
LIN {X 0,Y 363.092,Z 216.1,A -85,B 0,C 180,E1 -13172.16,E2 -13172.16} C_VEL
LIN {X 0,Y 363.27,Z 208.178,A -85,B 0,C 180,E1 -13175.479,E2 -13175.479} C_VEL
LIN {X 0,Y 362.667,Z 202.736,A -85,B 0,C 180,E1 -13177.826,E2 -13177.826} C_VEL
LIN {X 0,Y 361.953,Z 198.4,A -85,B 0,C 180,E1 -13179.732,E2 -13179.732} C_VEL
LIN {X 0,Y 361.841,Z 198.415,A -85,B 0,C 180,E1 -13182.828,E2 -13182.828} C_VEL
LIN {X 0,Y 361.824,Z 198.417,A -85,B 0,C 180,E1 -13185.946,E2 -13185.946} C_VEL
LIN {X 0,Y 361.839,Z 198.414,A -85,B 0,C 180,E1 -13189.244,E2 -13189.244} C_VEL
LIN {X 0,Y 361.867,Z 198.413,A -85,B 0,C 180,E1 -13192.981,E2 -13192.981} C_VEL
LIN {X 0,Y 361.861,Z 198.413,A -85,B 0,C 180,E1 -13196.631,E2 -13196.631} C_VEL
LIN {X 0,Y 361.783,Z 198.465,A -85,B 0,C 180,E1 -13199.662,E2 -13199.662} C_VEL
LIN {X 0,Y 361.843,Z 201.317,A -85,B 0,C 180,E1 -13202.214,E2 -13202.214} C_VEL
LIN {X 0,Y 361.784,Z 204.18,A -85,B 0,C 180,E1 -13204.698,E2 -13204.698} C_VEL
LIN {X 0,Y 361.661,Z 208.517,A -85,B 0,C 180,E1 -13208.331,E2 -13208.331} C_VEL
LIN {X 0,Y 361.656,Z 213.423,A -85,B 0,C 180,E1 -13212.216,E2 -13212.216} C_VEL
LIN {X 0,Y 361.679,Z 219.323,A -85,B 0,C 180,E1 -13216.514,E2 -13216.514} C_VEL
LIN {X 0,Y 361.681,Z 219.738,A -85,B 0,C 180,E1 -13216.8,E2 -13216.8} C_VEL
LIN {X 0,Y 364.277,Z 230.151,A -85,B 0,C 180,E1 -13217.392,E2 -13217.392} C_VEL
LIN {X 0,Y 365.936,Z 239.236,A -85,B 0,C 180,E1 -13218.084,E2 -13218.084} C_VEL
LIN {X 0,Y 365.601,Z 248.179,A -85,B 0,C 180,E1 -13218.916,E2 -13218.916} C_VEL
LIN {X 0,Y 365.127,Z 255.219,A -85,B 0,C 180,E1 -13219.76,E2 -13219.76} C_VEL
LIN {X 0,Y 364.486,Z 262.332,A -85,B 0,C 180,E1 -13220.845,E2 -13220.845} C_VEL
LIN {X 0,Y 363.899,Z 267.975,A -85,B 0,C 180,E1 -13221.95,E2 -13221.95} C_VEL
LIN {X 0,Y 363.636,Z 271.352,A -85,B 0,C 180,E1 -13222.782,E2 -13222.782} C_VEL
LIN {X 0,Y 363.14,Z 275.062,A -85,B 0,C 180,E1 -13223.888,E2 -13223.888} C_VEL
LIN {X 0,Y 362.792,Z 279.107,A -85,B 0,C 180,E1 -13225.554,E2 -13225.554} C_VEL
LIN {X 0,Y 362.362,Z 281.009,A -85,B 0,C 180,E1 -13226.663,E2 -13226.663} C_VEL
LIN {X 0,Y 362.28,Z 282.292,A -85,B 0,C 180,E1 -13227.775,E2 -13227.775} C_VEL
LIN {X 0,Y 362.133,Z 283.064,A -85,B 0,C 180,E1 -13228.887,E2 -13228.887} C_VEL
LIN {X 0,Y 362.072,Z 283.329,A -85,B 0,C 180,E1 -13229.999,E2 -13229.999} C_VEL
LIN {X 0,Y 362.129,Z 283.103,A -85,B 0,C 180,E1 -13231.111,E2 -13231.111} C_VEL
LIN {X 0,Y 362.271,Z 282.384,A -85,B 0,C 180,E1 -13232.222,E2 -13232.222} C_VEL
LIN {X 0,Y 362.358,Z 281.157,A -85,B 0,C 180,E1 -13233.334,E2 -13233.334} C_VEL
LIN {X 0,Y 363,Z 278.161,A -85,B 0,C 180,E1 -13234.997,E2 -13234.997} C_VEL
LIN {X 0,Y 363.213,Z 273.692,A -85,B 0,C 180,E1 -13236.665,E2 -13236.665} C_VEL
LIN {X 0,Y 363.71,Z 270.715,A -85,B 0,C 180,E1 -13237.493,E2 -13237.493} C_VEL
LIN {X 0,Y 364.035,Z 267.144,A -85,B 0,C 180,E1 -13238.324,E2 -13238.324} C_VEL
LIN {X 0,Y 364.657,Z 261.295,A -85,B 0,C 180,E1 -13239.427,E2 -13239.427} C_VEL
LIN {X 0,Y 365.111,Z 256.218,A -85,B 0,C 180,E1 -13240.206,E2 -13240.206} C_VEL
LIN {X 0,Y 365.505,Z 249.146,A -85,B 0,C 180,E1 -13241.084,E2 -13241.084} C_VEL
LIN {X 0,Y 366.003,Z 240.833,A -85,B 0,C 180,E1 -13241.883,E2 -13241.883} C_VEL
LIN {X 0,Y 365.657,Z 236.981,A -85,B 0,C 180,E1 -13242.204,E2 -13242.204} C_VEL
LIN {X 0,Y 363.592,Z 227.136,A -85,B 0,C 180,E1 -13242.903,E2 -13242.903} C_VEL
LIN {X 0,Y 361.685,Z 219.698,A -85,B 0,C 180,E1 -13243.339,E2 -13243.339} C_VEL
LIN {X 0,Y 361.62,Z 214.708,A -85,B 0,C 180,E1 -13246.947,E2 -13246.947} C_VEL
LIN {X 0,Y 361.656,Z 210.163,A -85,B 0,C 180,E1 -13250.473,E2 -13250.473} C_VEL
LIN {X 0,Y 361.766,Z 205.797,A -85,B 0,C 180,E1 -13254.075,E2 -13254.075} C_VEL
LIN {X 0,Y 361.846,Z 202.754,A -85,B 0,C 180,E1 -13256.691,E2 -13256.691} C_VEL
LIN {X 0,Y 361.829,Z 200.824,A -85,B 0,C 180,E1 -13258.346,E2 -13258.346} C_VEL
LIN {X 0,Y 361.145,Z 199.983,A -85,B 0,C 180,E1 -13259.266,E2 -13259.266} C_VEL
LIN {X 0,Y 358.259,Z 199.353,A -85,B 0,C 180,E1 -13260.774,E2 -13260.774} C_VEL
LIN {X 0,Y 355.842,Z 199.269,A -85,B 0,C 180,E1 -13262,E2 -13262} C_VEL
LIN {X 0,Y 354.839,Z 199.289,A -85,B 0,C 180,E1 -13262.949,E2 -13262.949} C_VEL
LIN {X 0,Y 354.775,Z 199.292,A -85,B 0,C 180,E1 -13263.27,E2 -13263.27} C_VEL
LIN {X 0,Y 354.796,Z 199.289,A -85,B 0,C 180,E1 -13266.457,E2 -13266.457} C_VEL
LIN {X 0,Y 354.818,Z 199.288,A -85,B 0,C 180,E1 -13269.422,E2 -13269.422} C_VEL
LIN {X 0,Y 354.782,Z 199.294,A -85,B 0,C 180,E1 -13272.866,E2 -13272.866} C_VEL
LIN {X 0,Y 354.768,Z 199.291,A -85,B 0,C 180,E1 -13276.103,E2 -13276.103} C_VEL
LIN {X 0,Y 354.781,Z 199.288,A -85,B 0,C 180,E1 -13279.178,E2 -13279.178} C_VEL
LIN {X 0,Y 354.8,Z 199.287,A -85,B 0,C 180,E1 -13282.401,E2 -13282.401} C_VEL
LIN {X 0,Y 354.804,Z 199.288,A -85,B 0,C 180,E1 -13284.94,E2 -13284.94} C_VEL
LIN {X 0,Y 354.806,Z 199.292,A -85,B 0,C 180,E1 -13288.398,E2 -13288.398} C_VEL
LIN {X 0,Y 354.845,Z 199.28,A -85,B 0,C 180,E1 -13291.618,E2 -13291.618} C_VEL
LIN {X 0,Y 354.89,Z 199.273,A -85,B 0,C 180,E1 -13294.172,E2 -13294.172} C_VEL
LIN {X 0,Y 354.824,Z 199.288,A -85,B 0,C 180,E1 -13297.893,E2 -13297.893} C_VEL
LIN {X 0,Y 354.913,Z 199.278,A -85,B 0,C 180,E1 -13301.89,E2 -13301.89} C_VEL
LIN {X 0,Y 354.932,Z 199.27,A -85,B 0,C 180,E1 -13305.98,E2 -13305.98} C_VEL
LIN {X 0,Y 354.967,Z 199.258,A -85,B 0,C 180,E1 -13309.735,E2 -13309.735} C_VEL
LIN {X 0,Y 355.112,Z 199.251,A -85,B 0,C 180,E1 -13313.18,E2 -13313.18} C_VEL
LIN {X 0,Y 355.234,Z 199.233,A -85,B 0,C 180,E1 -13317.732,E2 -13317.732} C_VEL
LIN {X 0,Y 355.385,Z 199.204,A -85,B 0,C 180,E1 -13320,E2 -13320} C_VEL
LIN {X 0,Y 355.23,Z 199.234,A -85,B 0,C 180,E1 -13322.268,E2 -13322.268} C_VEL
LIN {X 0,Y 355.125,Z 199.251,A -85,B 0,C 180,E1 -13326.819,E2 -13326.819} C_VEL
LIN {X 0,Y 355.003,Z 199.256,A -85,B 0,C 180,E1 -13329.113,E2 -13329.113} C_VEL
LIN {X 0,Y 354.909,Z 199.272,A -85,B 0,C 180,E1 -13332.581,E2 -13332.581} C_VEL
LIN {X 0,Y 354.875,Z 199.282,A -85,B 0,C 180,E1 -13336.097,E2 -13336.097} C_VEL
LIN {X 0,Y 354.83,Z 199.288,A -85,B 0,C 180,E1 -13339.677,E2 -13339.677} C_VEL
LIN {X 0,Y 354.798,Z 199.291,A -85,B 0,C 180,E1 -13343.339,E2 -13343.339} C_VEL
LIN {X 0,Y 354.782,Z 199.293,A -85,B 0,C 180,E1 -13347.105,E2 -13347.105} C_VEL
LIN {X 0,Y 354.785,Z 199.294,A -85,B 0,C 180,E1 -13349.685,E2 -13349.685} C_VEL
LIN {X 0,Y 354.777,Z 199.291,A -85,B 0,C 180,E1 -13352.334,E2 -13352.334} C_VEL
LIN {X 0,Y 354.812,Z 199.291,A -85,B 0,C 180,E1 -13355.7,E2 -13355.7} C_VEL
LIN {X 0,Y 354.759,Z 199.291,A -85,B 0,C 180,E1 -13359.414,E2 -13359.414} C_VEL
LIN {X 0,Y 354.777,Z 199.297,A -85,B 0,C 180,E1 -13362.868,E2 -13362.868} C_VEL
LIN {X 0,Y 354.76,Z 199.296,A -85,B 0,C 180,E1 -13366.105,E2 -13366.105} C_VEL
LIN {X 0,Y 354.817,Z 199.373,A -85,B 0,C 180,E1 -13367.237,E2 -13367.237} C_VEL
LIN {X 0,Y 357.093,Z 208.738,A -85,B 0,C 180,E1 -13370.777,E2 -13370.777} C_VEL
LIN {X 0,Y 359.291,Z 218.285,A -85,B 0,C 180,E1 -13374.07,E2 -13374.07} C_VEL
LIN {X 0,Y 361.501,Z 228.653,A -85,B 0,C 180,E1 -13377.353,E2 -13377.353} C_VEL
LIN {X 0,Y 361.638,Z 232.092,A -85,B 0,C 180,E1 -13378.353,E2 -13378.353} C_VEL
LIN {X 0,Y 359.108,Z 246.832,A -85,B 0,C 180,E1 -13382.304,E2 -13382.304} C_VEL
LIN {X 0,Y 357.095,Z 261.448,A -85,B 0,C 180,E1 -13386.207,E2 -13386.207} C_VEL
LIN {X 0,Y 355.427,Z 276.721,A -85,B 0,C 180,E1 -13390.359,E2 -13390.359} C_VEL
LIN {X 0,Y 355.184,Z 279.046,A -85,B 0,C 180,E1 -13391.006,E2 -13391.006} C_VEL
LIN {X 0,Y 356.808,Z 298.874,A -85,B 0,C 180,E1 -13391.757,E2 -13391.757} C_VEL
LIN {X 0,Y 357.639,Z 311.097,A -85,B 0,C 180,E1 -13392.416,E2 -13392.416} C_VEL
LIN {X 0,Y 357.584,Z 321.807,A -85,B 0,C 180,E1 -13393.15,E2 -13393.15} C_VEL
LIN {X 0,Y 356.66,Z 333.36,A -85,B 0,C 180,E1 -13394.135,E2 -13394.135} C_VEL
LIN {X 0,Y 355.888,Z 344.242,A -85,B 0,C 180,E1 -13395.297,E2 -13395.297} C_VEL
LIN {X 0,Y 355.231,Z 353.855,A -85,B 0,C 180,E1 -13396.559,E2 -13396.559} C_VEL
LIN {X 0,Y 354.578,Z 362.798,A -85,B 0,C 180,E1 -13397.99,E2 -13397.99} C_VEL
LIN {X 0,Y 353.993,Z 371.566,A -85,B 0,C 180,E1 -13399.709,E2 -13399.709} C_VEL
LIN {X 0,Y 353.691,Z 378.565,A -85,B 0,C 180,E1 -13401.431,E2 -13401.431} C_VEL
LIN {X 0,Y 353.543,Z 384.122,A -85,B 0,C 180,E1 -13403.151,E2 -13403.151} C_VEL
LIN {X 0,Y 353.548,Z 388.426,A -85,B 0,C 180,E1 -13404.869,E2 -13404.869} C_VEL
LIN {X 0,Y 353.498,Z 391.571,A -85,B 0,C 180,E1 -13406.582,E2 -13406.582} C_VEL
LIN {X 0,Y 353.608,Z 393.105,A -85,B 0,C 180,E1 -13407.723,E2 -13407.723} C_VEL
LIN {X 0,Y 353.587,Z 394.158,A -85,B 0,C 180,E1 -13408.863,E2 -13408.863} C_VEL
LIN {X 0,Y 353.605,Z 394.76,A -85,B 0,C 180,E1 -13410.001,E2 -13410.001} C_VEL
LIN {X 0,Y 353.568,Z 394.943,A -85,B 0,C 180,E1 -13411.14,E2 -13411.14} C_VEL
LIN {X 0,Y 353.501,Z 394.701,A -85,B 0,C 180,E1 -13412.28,E2 -13412.28} C_VEL
LIN {X 0,Y 353.405,Z 393.99,A -85,B 0,C 180,E1 -13413.422,E2 -13413.422} C_VEL
LIN {X 0,Y 353.432,Z 392.87,A -85,B 0,C 180,E1 -13414.564,E2 -13414.564} C_VEL
LIN {X 0,Y 353.398,Z 390.701,A -85,B 0,C 180,E1 -13416.094,E2 -13416.094} C_VEL
LIN {X 0,Y 353.631,Z 386.896,A -85,B 0,C 180,E1 -13417.998,E2 -13417.998} C_VEL
LIN {X 0,Y 354.018,Z 382.33,A -85,B 0,C 180,E1 -13419.716,E2 -13419.716} C_VEL
LIN {X 0,Y 354.785,Z 375.558,A -85,B 0,C 180,E1 -13421.716,E2 -13421.716} C_VEL
LIN {X 0,Y 356.119,Z 366.892,A -85,B 0,C 180,E1 -13423.7,E2 -13423.7} C_VEL
LIN {X 0,Y 357.328,Z 357.309,A -85,B 0,C 180,E1 -13425.476,E2 -13425.476} C_VEL
LIN {X 0,Y 359.157,Z 346.499,A -85,B 0,C 180,E1 -13427.07,E2 -13427.07} C_VEL
LIN {X 0,Y 360.955,Z 334.951,A -85,B 0,C 180,E1 -13428.446,E2 -13428.446} C_VEL
LIN {X 0,Y 362.786,Z 322.167,A -85,B 0,C 180,E1 -13429.671,E2 -13429.671} C_VEL
LIN {X 0,Y 363.439,Z 308.736,A -85,B 0,C 180,E1 -13430.768,E2 -13430.768} C_VEL
LIN {X 0,Y 362.808,Z 294.65,A -85,B 0,C 180,E1 -13431.788,E2 -13431.788} C_VEL
LIN {X 0,Y 360.641,Z 280.216,A -85,B 0,C 180,E1 -13432.779,E2 -13432.779} C_VEL
LIN {X 0,Y 359.433,Z 274.361,A -85,B 0,C 180,E1 -13433.221,E2 -13433.221} C_VEL
LIN {X 0,Y 359.043,Z 263.1,A -85,B 0,C 180,E1 -13434.829,E2 -13434.829} C_VEL
LIN {X 0,Y 358.916,Z 255.147,A -85,B 0,C 180,E1 -13436.141,E2 -13436.141} C_VEL
LIN {X 0,Y 359.167,Z 246.494,A -85,B 0,C 180,E1 -13437.773,E2 -13437.773} C_VEL
LIN {X 0,Y 361.625,Z 231.978,A -85,B 0,C 180,E1 -13441.651,E2 -13441.651} C_VEL
LIN {X 0,Y 361.414,Z 228.512,A -85,B 0,C 180,E1 -13442.659,E2 -13442.659} C_VEL
LIN {X 0,Y 360.589,Z 224.65,A -85,B 0,C 180,E1 -13443.912,E2 -13443.912} C_VEL
LIN {X 0,Y 360.659,Z 221.305,A -85,B 0,C 180,E1 -13445.776,E2 -13445.776} C_VEL
LIN {X 0,Y 361.239,Z 217.594,A -85,B 0,C 180,E1 -13448.903,E2 -13448.903} C_VEL
LIN {X 0,Y 361.502,Z 217.002,A -85,B 0,C 180,E1 -13449.909,E2 -13449.909} C_VEL
LIN {X 0,Y 361.31,Z 216.977,A -85,B 0,C 180,E1 -13452.34,E2 -13452.34} C_VEL
LIN {X 0,Y 361.3,Z 217.699,A -85,B 0,C 180,E1 -13454.45,E2 -13454.45} C_VEL
LIN {X 0,Y 361.519,Z 220.092,A -85,B 0,C 180,E1 -13457.625,E2 -13457.625} C_VEL
LIN {X 0,Y 361.98,Z 223.872,A -85,B 0,C 180,E1 -13460.953,E2 -13460.953} C_VEL
LIN {X 0,Y 362.172,Z 226.844,A -85,B 0,C 180,E1 -13463.018,E2 -13463.018} C_VEL
LIN {X 0,Y 361.826,Z 229.72,A -85,B 0,C 180,E1 -13464.668,E2 -13464.668} C_VEL
LIN {X 0,Y 360.08,Z 238.645,A -85,B 0,C 180,E1 -13469.182,E2 -13469.182} C_VEL
LIN {X 0,Y 358.95,Z 246.968,A -85,B 0,C 180,E1 -13473.235,E2 -13473.235} C_VEL
LIN {X 0,Y 358.123,Z 254.511,A -85,B 0,C 180,E1 -13476.776,E2 -13476.776} C_VEL
LIN {X 0,Y 363.169,Z 268.524,A -85,B 0,C 180,E1 -13478.265,E2 -13478.265} C_VEL
LIN {X 0,Y 365.654,Z 278.557,A -85,B 0,C 180,E1 -13479.31,E2 -13479.31} C_VEL
LIN {X 0,Y 366.084,Z 281.581,A -85,B 0,C 180,E1 -13479.612,E2 -13479.612} C_VEL
LIN {X 0,Y 364.535,Z 294.414,A -85,B 0,C 180,E1 -13480.722,E2 -13480.722} C_VEL
LIN {X 0,Y 362.816,Z 305.819,A -85,B 0,C 180,E1 -13481.945,E2 -13481.945} C_VEL
LIN {X 0,Y 361.179,Z 316.084,A -85,B 0,C 180,E1 -13483.321,E2 -13483.321} C_VEL
LIN {X 0,Y 359.651,Z 324.665,A -85,B 0,C 180,E1 -13484.704,E2 -13484.704} C_VEL
LIN {X 0,Y 358.131,Z 333.108,A -85,B 0,C 180,E1 -13486.38,E2 -13486.38} C_VEL
LIN {X 0,Y 356.97,Z 339.969,A -85,B 0,C 180,E1 -13488.07,E2 -13488.07} C_VEL
LIN {X 0,Y 355.909,Z 345.534,A -85,B 0,C 180,E1 -13489.763,E2 -13489.763} C_VEL
LIN {X 0,Y 355.097,Z 350.06,A -85,B 0,C 180,E1 -13491.521,E2 -13491.521} C_VEL
LIN {X 0,Y 354.361,Z 353.266,A -85,B 0,C 180,E1 -13493.166,E2 -13493.166} C_VEL
LIN {X 0,Y 354.227,Z 354.934,A -85,B 0,C 180,E1 -13494.307,E2 -13494.307} C_VEL
LIN {X 0,Y 354.097,Z 356.149,A -85,B 0,C 180,E1 -13495.446,E2 -13495.446} C_VEL
LIN {X 0,Y 353.65,Z 357.434,A -85,B 0,C 180,E1 -13497.722,E2 -13497.722} C_VEL
LIN {X 0,Y 353.514,Z 357.439,A -85,B 0,C 180,E1 -13498.861,E2 -13498.861} C_VEL
LIN {X 0,Y 353.455,Z 357.026,A -85,B 0,C 180,E1 -13500,E2 -13500} C_VEL
LIN {X 0,Y 353.463,Z 356.218,A -85,B 0,C 180,E1 -13501.139,E2 -13501.139} C_VEL
LIN {X 0,Y 353.478,Z 354.993,A -85,B 0,C 180,E1 -13502.279,E2 -13502.279} C_VEL
LIN {X 0,Y 353.528,Z 352.331,A -85,B 0,C 180,E1 -13503.99,E2 -13503.99} C_VEL
LIN {X 0,Y 353.698,Z 348.626,A -85,B 0,C 180,E1 -13505.702,E2 -13505.702} C_VEL
LIN {X 0,Y 353.96,Z 343.786,A -85,B 0,C 180,E1 -13507.415,E2 -13507.415} C_VEL
LIN {X 0,Y 354.453,Z 336.548,A -85,B 0,C 180,E1 -13509.415,E2 -13509.415} C_VEL
LIN {X 0,Y 355.048,Z 328.705,A -85,B 0,C 180,E1 -13511.128,E2 -13511.128} C_VEL
LIN {X 0,Y 355.832,Z 318.997,A -85,B 0,C 180,E1 -13512.838,E2 -13512.838} C_VEL
LIN {X 0,Y 356.566,Z 309.018,A -85,B 0,C 180,E1 -13514.263,E2 -13514.263} C_VEL
LIN {X 0,Y 357.393,Z 297.51,A -85,B 0,C 180,E1 -13515.597,E2 -13515.597} C_VEL
LIN {X 0,Y 358.192,Z 285.85,A -85,B 0,C 180,E1 -13516.676,E2 -13516.676} C_VEL
LIN {X 0,Y 358.933,Z 273.74,A -85,B 0,C 180,E1 -13517.557,E2 -13517.557} C_VEL
LIN {X 0,Y 356.84,Z 260.676,A -85,B 0,C 180,E1 -13518.368,E2 -13518.368} C_VEL
LIN {X 0,Y 354.831,Z 248.991,A -85,B 0,C 180,E1 -13518.93,E2 -13518.93} C_VEL
LIN {X 0,Y 355.163,Z 239.874,A -85,B 0,C 180,E1 -13522.698,E2 -13522.698} C_VEL
LIN {X 0,Y 355.473,Z 230.962,A -85,B 0,C 180,E1 -13526.414,E2 -13526.414} C_VEL
LIN {X 0,Y 355.815,Z 221.837,A -85,B 0,C 180,E1 -13530.243,E2 -13530.243} C_VEL
LIN {X 0,Y 356.103,Z 215.625,A -85,B 0,C 180,E1 -13532.87,E2 -13532.87} C_VEL
LIN {X 0,Y 356.275,Z 209.514,A -85,B 0,C 180,E1 -13535.445,E2 -13535.445} C_VEL
LIN {X 0,Y 355.721,Z 204.084,A -85,B 0,C 180,E1 -13537.787,E2 -13537.787} C_VEL
LIN {X 0,Y 354.896,Z 199.279,A -85,B 0,C 180,E1 -13540,E2 -13540} C_VEL
LIN {X 0,Y 354.773,Z 199.294,A -85,B 0,C 180,E1 -13543.896,E2 -13543.896} C_VEL
LIN {X 0,Y 354.8,Z 199.29,A -85,B 0,C 180,E1 -13547.662,E2 -13547.662} C_VEL
LIN {X 0,Y 354.79,Z 199.293,A -85,B 0,C 180,E1 -13550.661,E2 -13550.661} C_VEL
LIN {X 0,Y 354.823,Z 199.292,A -85,B 0,C 180,E1 -13554.301,E2 -13554.301} C_VEL
LIN {X 0,Y 354.773,Z 199.295,A -85,B 0,C 180,E1 -13557.664,E2 -13557.664} C_VEL
LIN {X 0,Y 354.76,Z 199.46,A -85,B 0,C 180,E1 -13559.491,E2 -13559.491} C_VEL
LIN {X 0,Y 354.845,Z 203.408,A -85,B 0,C 180,E1 -13563.033,E2 -13563.033} C_VEL
LIN {X 0,Y 354.74,Z 207.648,A -85,B 0,C 180,E1 -13566.656,E2 -13566.656} C_VEL
LIN {X 0,Y 354.603,Z 212.094,A -85,B 0,C 180,E1 -13570.309,E2 -13570.309} C_VEL
LIN {X 0,Y 354.629,Z 215.192,A -85,B 0,C 180,E1 -13572.705,E2 -13572.705} C_VEL
LIN {X 0,Y 354.667,Z 220.363,A -85,B 0,C 180,E1 -13576.474,E2 -13576.474} C_VEL
LIN {X 0,Y 357.274,Z 230.684,A -85,B 0,C 180,E1 -13577.076,E2 -13577.076} C_VEL
LIN {X 0,Y 358.9,Z 238.8,A -85,B 0,C 180,E1 -13577.703,E2 -13577.703} C_VEL
LIN {X 0,Y 358.942,Z 244.815,A -85,B 0,C 180,E1 -13578.235,E2 -13578.235} C_VEL
LIN {X 0,Y 358.449,Z 253.214,A -85,B 0,C 180,E1 -13579.136,E2 -13579.136} C_VEL
LIN {X 0,Y 357.931,Z 260.07,A -85,B 0,C 180,E1 -13580.106,E2 -13580.106} C_VEL
LIN {X 0,Y 357.379,Z 266.36,A -85,B 0,C 180,E1 -13581.232,E2 -13581.232} C_VEL
LIN {X 0,Y 356.796,Z 271.316,A -85,B 0,C 180,E1 -13582.358,E2 -13582.358} C_VEL
LIN {X 0,Y 356.262,Z 274.34,A -85,B 0,C 180,E1 -13583.201,E2 -13583.201} C_VEL
LIN {X 0,Y 356.011,Z 278.906,A -85,B 0,C 180,E1 -13584.902,E2 -13584.902} C_VEL
LIN {X 0,Y 355.349,Z 281.986,A -85,B 0,C 180,E1 -13586.597,E2 -13586.597} C_VEL
LIN {X 0,Y 355.259,Z 283.266,A -85,B 0,C 180,E1 -13587.731,E2 -13587.731} C_VEL
LIN {X 0,Y 355.109,Z 284.038,A -85,B 0,C 180,E1 -13588.865,E2 -13588.865} C_VEL
LIN {X 0,Y 355.046,Z 284.303,A -85,B 0,C 180,E1 -13589.999,E2 -13589.999} C_VEL
LIN {X 0,Y 355.105,Z 284.076,A -85,B 0,C 180,E1 -13591.133,E2 -13591.133} C_VEL
LIN {X 0,Y 355.251,Z 283.358,A -85,B 0,C 180,E1 -13592.266,E2 -13592.266} C_VEL
LIN {X 0,Y 355.345,Z 282.133,A -85,B 0,C 180,E1 -13593.4,E2 -13593.4} C_VEL
LIN {X 0,Y 356.002,Z 279.145,A -85,B 0,C 180,E1 -13595.095,E2 -13595.095} C_VEL
LIN {X 0,Y 356.233,Z 274.692,A -85,B 0,C 180,E1 -13596.797,E2 -13596.797} C_VEL
LIN {X 0,Y 356.745,Z 271.721,A -85,B 0,C 180,E1 -13597.64,E2 -13597.64} C_VEL
LIN {X 0,Y 357.086,Z 268.178,A -85,B 0,C 180,E1 -13598.487,E2 -13598.487} C_VEL
LIN {X 0,Y 357.742,Z 262.359,A -85,B 0,C 180,E1 -13599.611,E2 -13599.611} C_VEL
LIN {X 0,Y 358.215,Z 257.295,A -85,B 0,C 180,E1 -13600.409,E2 -13600.409} C_VEL
LIN {X 0,Y 358.619,Z 250.324,A -85,B 0,C 180,E1 -13601.3,E2 -13601.3} C_VEL
LIN {X 0,Y 359.082,Z 243.462,A -85,B 0,C 180,E1 -13602,E2 -13602} C_VEL
LIN {X 0,Y 359.171,Z 240.139,A -85,B 0,C 180,E1 -13602.284,E2 -13602.284} C_VEL
LIN {X 0,Y 357.133,Z 230.087,A -85,B 0,C 180,E1 -13603.071,E2 -13603.071} C_VEL
LIN {X 0,Y 354.664,Z 220.35,A -85,B 0,C 180,E1 -13603.646,E2 -13603.646} C_VEL
LIN {X 0,Y 354.656,Z 214.466,A -85,B 0,C 180,E1 -13607.975,E2 -13607.975} C_VEL
LIN {X 0,Y 354.668,Z 210.184,A -85,B 0,C 180,E1 -13611.355,E2 -13611.355} C_VEL
LIN {X 0,Y 354.758,Z 206.375,A -85,B 0,C 180,E1 -13614.582,E2 -13614.582} C_VEL
LIN {X 0,Y 354.84,Z 203.458,A -85,B 0,C 180,E1 -13617.098,E2 -13617.098} C_VEL
LIN {X 0,Y 354.761,Z 199.404,A -85,B 0,C 180,E1 -13620.67,E2 -13620.67} C_VEL
LIN {X 0,Y 354.775,Z 199.292,A -85,B 0,C 180,E1 -13623.27,E2 -13623.27} C_VEL
LIN {X 0,Y 354.16,Z 199.372,A -85,B 0,C 180,E1 -13624.217,E2 -13624.217} C_VEL
LIN {X 0,Y 351.339,Z 199.724,A -85,B 0,C 180,E1 -13625.758,E2 -13625.758} C_VEL
LIN {X 0,Y 348.908,Z 200.025,A -85,B 0,C 180,E1 -13627.005,E2 -13627.005} C_VEL
LIN {X 0,Y 347.848,Z 200.156,A -85,B 0,C 180,E1 -13627.97,E2 -13627.97} C_VEL
LIN {X 0,Y 347.755,Z 200.167,A -85,B 0,C 180,E1 -13628.297,E2 -13628.297} C_VEL
LIN {X 0,Y 347.745,Z 200.167,A -85,B 0,C 180,E1 -13631.829,E2 -13631.829} C_VEL
LIN {X 0,Y 347.759,Z 200.169,A -85,B 0,C 180,E1 -13635.015,E2 -13635.015} C_VEL
LIN {X 0,Y 347.743,Z 200.17,A -85,B 0,C 180,E1 -13638.396,E2 -13638.396} C_VEL
LIN {X 0,Y 347.767,Z 200.164,A -85,B 0,C 180,E1 -13642.01,E2 -13642.01} C_VEL
LIN {X 0,Y 347.736,Z 200.166,A -85,B 0,C 180,E1 -13645.535,E2 -13645.535} C_VEL
LIN {X 0,Y 347.755,Z 200.169,A -85,B 0,C 180,E1 -13648.301,E2 -13648.301} C_VEL
LIN {X 0,Y 347.797,Z 200.157,A -85,B 0,C 180,E1 -13650.989,E2 -13650.989} C_VEL
LIN {X 0,Y 347.823,Z 200.158,A -85,B 0,C 180,E1 -13653.607,E2 -13653.607} C_VEL
LIN {X 0,Y 347.778,Z 200.161,A -85,B 0,C 180,E1 -13656.161,E2 -13656.161} C_VEL
LIN {X 0,Y 347.807,Z 200.153,A -85,B 0,C 180,E1 -13659.909,E2 -13659.909} C_VEL
LIN {X 0,Y 347.857,Z 200.154,A -85,B 0,C 180,E1 -13662.359,E2 -13662.359} C_VEL
LIN {X 0,Y 347.886,Z 200.147,A -85,B 0,C 180,E1 -13665.97,E2 -13665.97} C_VEL
LIN {X 0,Y 347.918,Z 200.137,A -85,B 0,C 180,E1 -13669.525,E2 -13669.525} C_VEL
LIN {X 0,Y 348.079,Z 200.127,A -85,B 0,C 180,E1 -13673.042,E2 -13673.042} C_VEL
LIN {X 0,Y 348.196,Z 200.11,A -85,B 0,C 180,E1 -13677.686,E2 -13677.686} C_VEL
LIN {X 0,Y 348.334,Z 200.082,A -85,B 0,C 180,E1 -13680,E2 -13680} C_VEL
LIN {X 0,Y 348.193,Z 200.111,A -85,B 0,C 180,E1 -13682.314,E2 -13682.314} C_VEL
LIN {X 0,Y 348.093,Z 200.126,A -85,B 0,C 180,E1 -13686.958,E2 -13686.958} C_VEL
LIN {X 0,Y 347.916,Z 200.144,A -85,B 0,C 180,E1 -13690.475,E2 -13690.475} C_VEL
LIN {X 0,Y 347.887,Z 200.145,A -85,B 0,C 180,E1 -13694.15,E2 -13694.15} C_VEL
LIN {X 0,Y 347.817,Z 200.156,A -85,B 0,C 180,E1 -13698.26,E2 -13698.26} C_VEL
LIN {X 0,Y 347.756,Z 200.17,A -85,B 0,C 180,E1 -13701.627,E2 -13701.627} C_VEL
LIN {X 0,Y 347.728,Z 200.172,A -85,B 0,C 180,E1 -13705.115,E2 -13705.115} C_VEL
LIN {X 0,Y 347.718,Z 200.174,A -85,B 0,C 180,E1 -13707.702,E2 -13707.702} C_VEL
LIN {X 0,Y 347.728,Z 200.17,A -85,B 0,C 180,E1 -13710.35,E2 -13710.35} C_VEL
LIN {X 0,Y 347.739,Z 200.165,A -85,B 0,C 180,E1 -13714.045,E2 -13714.045} C_VEL
LIN {X 0,Y 347.747,Z 200.167,A -85,B 0,C 180,E1 -13717.323,E2 -13717.323} C_VEL
LIN {X 0,Y 347.733,Z 200.16,A -85,B 0,C 180,E1 -13721.602,E2 -13721.602} C_VEL
LIN {X 0,Y 347.698,Z 200.174,A -85,B 0,C 180,E1 -13725.028,E2 -13725.028} C_VEL
LIN {X 0,Y 347.749,Z 200.32,A -85,B 0,C 180,E1 -13726.598,E2 -13726.598} C_VEL
LIN {X 0,Y 349.921,Z 209.001,A -85,B 0,C 180,E1 -13730.009,E2 -13730.009} C_VEL
LIN {X 0,Y 352.184,Z 218.977,A -85,B 0,C 180,E1 -13733.584,E2 -13733.584} C_VEL
LIN {X 0,Y 354.399,Z 229.268,A -85,B 0,C 180,E1 -13736.954,E2 -13736.954} C_VEL
LIN {X 0,Y 354.81,Z 231.573,A -85,B 0,C 180,E1 -13737.671,E2 -13737.671} C_VEL
LIN {X 0,Y 354.513,Z 234.411,A -85,B 0,C 180,E1 -13738.479,E2 -13738.479} C_VEL
LIN {X 0,Y 352.024,Z 248.467,A -85,B 0,C 180,E1 -13742.345,E2 -13742.345} C_VEL
LIN {X 0,Y 349.982,Z 262.929,A -85,B 0,C 180,E1 -13746.322,E2 -13746.322} C_VEL
LIN {X 0,Y 348.171,Z 278.649,A -85,B 0,C 180,E1 -13750.737,E2 -13750.737} C_VEL
LIN {X 0,Y 349.862,Z 299.969,A -85,B 0,C 180,E1 -13751.601,E2 -13751.601} C_VEL
LIN {X 0,Y 350.635,Z 313.162,A -85,B 0,C 180,E1 -13752.37,E2 -13752.37} C_VEL
LIN {X 0,Y 350.599,Z 321.332,A -85,B 0,C 180,E1 -13752.954,E2 -13752.954} C_VEL
LIN {X 0,Y 349.582,Z 334.363,A -85,B 0,C 180,E1 -13754.104,E2 -13754.104} C_VEL
LIN {X 0,Y 348.751,Z 345.082,A -85,B 0,C 180,E1 -13755.306,E2 -13755.306} C_VEL
LIN {X 0,Y 348.096,Z 354.32,A -85,B 0,C 180,E1 -13756.576,E2 -13756.576} C_VEL
LIN {X 0,Y 347.479,Z 363.12,A -85,B 0,C 180,E1 -13758.037,E2 -13758.037} C_VEL
LIN {X 0,Y 346.888,Z 371.734,A -85,B 0,C 180,E1 -13759.79,E2 -13759.79} C_VEL
LIN {X 0,Y 346.603,Z 378.602,A -85,B 0,C 180,E1 -13761.548,E2 -13761.548} C_VEL
LIN {X 0,Y 346.476,Z 383.254,A -85,B 0,C 180,E1 -13763.011,E2 -13763.011} C_VEL
LIN {X 0,Y 346.474,Z 387.661,A -85,B 0,C 180,E1 -13764.764,E2 -13764.764} C_VEL
LIN {X 0,Y 346.414,Z 390.906,A -85,B 0,C 180,E1 -13766.512,E2 -13766.512} C_VEL
LIN {X 0,Y 346.542,Z 392.487,A -85,B 0,C 180,E1 -13767.677,E2 -13767.677} C_VEL
LIN {X 0,Y 346.52,Z 393.619,A -85,B 0,C 180,E1 -13768.839,E2 -13768.839} C_VEL
LIN {X 0,Y 346.534,Z 394.274,A -85,B 0,C 180,E1 -13770.001,E2 -13770.001} C_VEL
LIN {X 0,Y 346.499,Z 394.5,A -85,B 0,C 180,E1 -13771.164,E2 -13771.164} C_VEL
LIN {X 0,Y 346.402,Z 394.308,A -85,B 0,C 180,E1 -13772.327,E2 -13772.327} C_VEL
LIN {X 0,Y 346.32,Z 393.682,A -85,B 0,C 180,E1 -13773.492,E2 -13773.492} C_VEL
LIN {X 0,Y 346.338,Z 392.608,A -85,B 0,C 180,E1 -13774.657,E2 -13774.657} C_VEL
LIN {X 0,Y 346.326,Z 390.748,A -85,B 0,C 180,E1 -13776.088,E2 -13776.088} C_VEL
LIN {X 0,Y 346.57,Z 386.84,A -85,B 0,C 180,E1 -13778.162,E2 -13778.162} C_VEL
LIN {X 0,Y 347,Z 382.403,A -85,B 0,C 180,E1 -13779.915,E2 -13779.915} C_VEL
LIN {X 0,Y 347.838,Z 375.777,A -85,B 0,C 180,E1 -13781.954,E2 -13781.954} C_VEL
LIN {X 0,Y 349.043,Z 368.692,A -85,B 0,C 180,E1 -13783.687,E2 -13783.687} C_VEL
LIN {X 0,Y 350.334,Z 359.279,A -85,B 0,C 180,E1 -13785.564,E2 -13785.564} C_VEL
LIN {X 0,Y 352.094,Z 349.57,A -85,B 0,C 180,E1 -13787.124,E2 -13787.124} C_VEL
LIN {X 0,Y 354.142,Z 337.662,A -85,B 0,C 180,E1 -13788.664,E2 -13788.664} C_VEL
LIN {X 0,Y 356.116,Z 325.736,A -85,B 0,C 180,E1 -13789.904,E2 -13789.904} C_VEL
LIN {X 0,Y 357.19,Z 312.868,A -85,B 0,C 180,E1 -13791.047,E2 -13791.047} C_VEL
LIN {X 0,Y 357.108,Z 300.379,A -85,B 0,C 180,E1 -13792.037,E2 -13792.037} C_VEL
LIN {X 0,Y 355.871,Z 288.097,A -85,B 0,C 180,E1 -13792.945,E2 -13792.945} C_VEL
LIN {X 0,Y 353.276,Z 273.955,A -85,B 0,C 180,E1 -13794.029,E2 -13794.029} C_VEL
LIN {X 0,Y 353.003,Z 263.511,A -85,B 0,C 180,E1 -13795.645,E2 -13795.645} C_VEL
LIN {X 0,Y 353.047,Z 256.177,A -85,B 0,C 180,E1 -13796.929,E2 -13796.929} C_VEL
LIN {X 0,Y 353.414,Z 248.207,A -85,B 0,C 180,E1 -13798.508,E2 -13798.508} C_VEL
LIN {X 0,Y 354.324,Z 238.758,A -85,B 0,C 180,E1 -13800.715,E2 -13800.715} C_VEL
LIN {X 0,Y 355.256,Z 233.105,A -85,B 0,C 180,E1 -13802.287,E2 -13802.287} C_VEL
LIN {X 0,Y 355.057,Z 228.494,A -85,B 0,C 180,E1 -13804.343,E2 -13804.343} C_VEL
LIN {X 0,Y 355.033,Z 224.838,A -85,B 0,C 180,E1 -13806.433,E2 -13806.433} C_VEL
LIN {X 0,Y 355.636,Z 221.688,A -85,B 0,C 180,E1 -13809.227,E2 -13809.227} C_VEL
LIN {X 0,Y 355.739,Z 221,A -85,B 0,C 180,E1 -13810.69,E2 -13810.69} C_VEL
LIN {X 0,Y 355.423,Z 221.421,A -85,B 0,C 180,E1 -13813.796,E2 -13813.796} C_VEL
LIN {X 0,Y 355.458,Z 223.358,A -85,B 0,C 180,E1 -13817.018,E2 -13817.018} C_VEL
LIN {X 0,Y 355.612,Z 225.513,A -85,B 0,C 180,E1 -13819.293,E2 -13819.293} C_VEL
LIN {X 0,Y 355.803,Z 227.227,A -85,B 0,C 180,E1 -13820.796,E2 -13820.796} C_VEL
LIN {X 0,Y 355.869,Z 230.133,A -85,B 0,C 180,E1 -13822.962,E2 -13822.962} C_VEL
LIN {X 0,Y 355.648,Z 232.011,A -85,B 0,C 180,E1 -13824.118,E2 -13824.118} C_VEL
LIN {X 0,Y 353.856,Z 239.722,A -85,B 0,C 180,E1 -13828.243,E2 -13828.243} C_VEL
LIN {X 0,Y 352.595,Z 247.286,A -85,B 0,C 180,E1 -13832.069,E2 -13832.069} C_VEL
LIN {X 0,Y 351.833,Z 253.687,A -85,B 0,C 180,E1 -13835.198,E2 -13835.198} C_VEL
LIN {X 0,Y 351.691,Z 255.445,A -85,B 0,C 180,E1 -13835.95,E2 -13835.95} C_VEL
LIN {X 0,Y 356.238,Z 267.586,A -85,B 0,C 180,E1 -13837.34,E2 -13837.34} C_VEL
LIN {X 0,Y 359.042,Z 277.876,A -85,B 0,C 180,E1 -13838.492,E2 -13838.492} C_VEL
LIN {X 0,Y 359.954,Z 283.948,A -85,B 0,C 180,E1 -13839.148,E2 -13839.148} C_VEL
LIN {X 0,Y 358.281,Z 296.168,A -85,B 0,C 180,E1 -13840.252,E2 -13840.252} C_VEL
LIN {X 0,Y 356.325,Z 308.095,A -85,B 0,C 180,E1 -13841.604,E2 -13841.604} C_VEL
LIN {X 0,Y 354.602,Z 318.027,A -85,B 0,C 180,E1 -13843.002,E2 -13843.002} C_VEL
LIN {X 0,Y 352.654,Z 327.795,A -85,B 0,C 180,E1 -13844.689,E2 -13844.689} C_VEL
LIN {X 0,Y 351.076,Z 335.746,A -85,B 0,C 180,E1 -13846.396,E2 -13846.396} C_VEL
LIN {X 0,Y 350.127,Z 341.176,A -85,B 0,C 180,E1 -13847.833,E2 -13847.833} C_VEL
LIN {X 0,Y 349.017,Z 346.587,A -85,B 0,C 180,E1 -13849.559,E2 -13849.559} C_VEL
LIN {X 0,Y 348.146,Z 350.959,A -85,B 0,C 180,E1 -13851.35,E2 -13851.35} C_VEL
LIN {X 0,Y 347.359,Z 354.053,A -85,B 0,C 180,E1 -13853.027,E2 -13853.027} C_VEL
LIN {X 0,Y 347.18,Z 355.611,A -85,B 0,C 180,E1 -13854.191,E2 -13854.191} C_VEL
LIN {X 0,Y 347.063,Z 356.762,A -85,B 0,C 180,E1 -13855.354,E2 -13855.354} C_VEL
LIN {X 0,Y 346.811,Z 357.542,A -85,B 0,C 180,E1 -13856.515,E2 -13856.515} C_VEL
LIN {X 0,Y 346.595,Z 357.907,A -85,B 0,C 180,E1 -13857.676,E2 -13857.676} C_VEL
LIN {X 0,Y 346.453,Z 357.836,A -85,B 0,C 180,E1 -13858.838,E2 -13858.838} C_VEL
LIN {X 0,Y 346.392,Z 357.369,A -85,B 0,C 180,E1 -13860,E2 -13860} C_VEL
LIN {X 0,Y 346.384,Z 356.505,A -85,B 0,C 180,E1 -13861.163,E2 -13861.163} C_VEL
LIN {X 0,Y 346.381,Z 355.182,A -85,B 0,C 180,E1 -13862.326,E2 -13862.326} C_VEL
LIN {X 0,Y 346.455,Z 352.41,A -85,B 0,C 180,E1 -13864.071,E2 -13864.071} C_VEL
LIN {X 0,Y 346.612,Z 348.594,A -85,B 0,C 180,E1 -13865.819,E2 -13865.819} C_VEL
LIN {X 0,Y 346.891,Z 343.638,A -85,B 0,C 180,E1 -13867.567,E2 -13867.567} C_VEL
LIN {X 0,Y 347.317,Z 337.414,A -85,B 0,C 180,E1 -13869.316,E2 -13869.316} C_VEL
LIN {X 0,Y 347.914,Z 329.705,A -85,B 0,C 180,E1 -13871.064,E2 -13871.064} C_VEL
LIN {X 0,Y 348.678,Z 320.098,A -85,B 0,C 180,E1 -13872.81,E2 -13872.81} C_VEL
LIN {X 0,Y 349.436,Z 310.325,A -85,B 0,C 180,E1 -13874.263,E2 -13874.263} C_VEL
LIN {X 0,Y 350.174,Z 301.253,A -85,B 0,C 180,E1 -13875.379,E2 -13875.379} C_VEL
LIN {X 0,Y 350.995,Z 289.324,A -85,B 0,C 180,E1 -13876.579,E2 -13876.579} C_VEL
LIN {X 0,Y 351.832,Z 277.07,A -85,B 0,C 180,E1 -13877.554,E2 -13877.554} C_VEL
LIN {X 0,Y 351.86,Z 273.591,A -85,B 0,C 180,E1 -13877.791,E2 -13877.791} C_VEL
LIN {X 0,Y 349.63,Z 260.159,A -85,B 0,C 180,E1 -13878.631,E2 -13878.631} C_VEL
LIN {X 0,Y 347.772,Z 249.324,A -85,B 0,C 180,E1 -13879.161,E2 -13879.161} C_VEL
LIN {X 0,Y 348.089,Z 241.178,A -85,B 0,C 180,E1 -13882.558,E2 -13882.558} C_VEL
LIN {X 0,Y 348.377,Z 233.692,A -85,B 0,C 180,E1 -13885.705,E2 -13885.705} C_VEL
LIN {X 0,Y 348.736,Z 224.878,A -85,B 0,C 180,E1 -13889.433,E2 -13889.433} C_VEL
LIN {X 0,Y 349.106,Z 216.655,A -85,B 0,C 180,E1 -13892.926,E2 -13892.926} C_VEL
LIN {X 0,Y 349.246,Z 210.167,A -85,B 0,C 180,E1 -13895.703,E2 -13895.703} C_VEL
LIN {X 0,Y 348.616,Z 204.595,A -85,B 0,C 180,E1 -13898.164,E2 -13898.164} C_VEL
LIN {X 0,Y 347.832,Z 200.159,A -85,B 0,C 180,E1 -13900.154,E2 -13900.154} C_VEL
LIN {X 0,Y 347.729,Z 200.171,A -85,B 0,C 180,E1 -13903.408,E2 -13903.408} C_VEL
LIN {X 0,Y 347.731,Z 200.17,A -85,B 0,C 180,E1 -13906.686,E2 -13906.686} C_VEL
LIN {X 0,Y 347.734,Z 200.172,A -85,B 0,C 180,E1 -13910.176,E2 -13910.176} C_VEL
LIN {X 0,Y 347.761,Z 200.17,A -85,B 0,C 180,E1 -13912.678,E2 -13912.678} C_VEL
LIN {X 0,Y 347.753,Z 200.17,A -85,B 0,C 180,E1 -13915.956,E2 -13915.956} C_VEL
LIN {X 0,Y 347.729,Z 200.277,A -85,B 0,C 180,E1 -13919.144,E2 -13919.144} C_VEL
LIN {X 0,Y 347.825,Z 203.774,A -85,B 0,C 180,E1 -13922.306,E2 -13922.306} C_VEL
LIN {X 0,Y 347.767,Z 207.322,A -85,B 0,C 180,E1 -13925.423,E2 -13925.423} C_VEL
LIN {X 0,Y 347.634,Z 211.193,A -85,B 0,C 180,E1 -13928.659,E2 -13928.659} C_VEL
LIN {X 0,Y 347.625,Z 215.824,A -85,B 0,C 180,E1 -13932.345,E2 -13932.345} C_VEL
LIN {X 0,Y 347.654,Z 221.087,A -85,B 0,C 180,E1 -13936.148,E2 -13936.148} C_VEL
LIN {X 0,Y 350.249,Z 231.03,A -85,B 0,C 180,E1 -13936.735,E2 -13936.735} C_VEL
LIN {X 0,Y 352.079,Z 240.17,A -85,B 0,C 180,E1 -13937.46,E2 -13937.46} C_VEL
LIN {X 0,Y 351.984,Z 247.979,A -85,B 0,C 180,E1 -13938.185,E2 -13938.185} C_VEL
LIN {X 0,Y 351.436,Z 256.342,A -85,B 0,C 180,E1 -13939.198,E2 -13939.198} C_VEL
LIN {X 0,Y 350.837,Z 262.804,A -85,B 0,C 180,E1 -13940.195,E2 -13940.195} C_VEL
LIN {X 0,Y 350.184,Z 268.744,A -85,B 0,C 180,E1 -13941.341,E2 -13941.341} C_VEL
LIN {X 0,Y 349.701,Z 273.371,A -85,B 0,C 180,E1 -13942.492,E2 -13942.492} C_VEL
LIN {X 0,Y 349.169,Z 277.053,A -85,B 0,C 180,E1 -13943.643,E2 -13943.643} C_VEL
LIN {X 0,Y 348.79,Z 281.07,A -85,B 0,C 180,E1 -13945.376,E2 -13945.376} C_VEL
LIN {X 0,Y 348.336,Z 282.962,A -85,B 0,C 180,E1 -13946.528,E2 -13946.528} C_VEL
LIN {X 0,Y 348.239,Z 284.24,A -85,B 0,C 180,E1 -13947.685,E2 -13947.685} C_VEL
LIN {X 0,Y 348.084,Z 285.011,A -85,B 0,C 180,E1 -13948.842,E2 -13948.842} C_VEL
LIN {X 0,Y 348.02,Z 285.277,A -85,B 0,C 180,E1 -13949.999,E2 -13949.999} C_VEL
LIN {X 0,Y 348.081,Z 285.05,A -85,B 0,C 180,E1 -13951.155,E2 -13951.155} C_VEL
LIN {X 0,Y 348.232,Z 284.332,A -85,B 0,C 180,E1 -13952.312,E2 -13952.312} C_VEL
LIN {X 0,Y 348.332,Z 283.109,A -85,B 0,C 180,E1 -13953.469,E2 -13953.469} C_VEL
LIN {X 0,Y 349.005,Z 280.128,A -85,B 0,C 180,E1 -13955.198,E2 -13955.198} C_VEL
LIN {X 0,Y 349.255,Z 275.69,A -85,B 0,C 180,E1 -13956.933,E2 -13956.933} C_VEL
LIN {X 0,Y 349.782,Z 272.725,A -85,B 0,C 180,E1 -13957.793,E2 -13957.793} C_VEL
LIN {X 0,Y 350.14,Z 269.211,A -85,B 0,C 180,E1 -13958.657,E2 -13958.657} C_VEL
LIN {X 0,Y 350.831,Z 263.422,A -85,B 0,C 180,E1 -13959.802,E2 -13959.802} C_VEL
LIN {X 0,Y 351.325,Z 258.31,A -85,B 0,C 180,E1 -13960.629,E2 -13960.629} C_VEL
LIN {X 0,Y 351.769,Z 251.494,A -85,B 0,C 180,E1 -13961.523,E2 -13961.523} C_VEL
LIN {X 0,Y 352.224,Z 244.725,A -85,B 0,C 180,E1 -13962.238,E2 -13962.238} C_VEL
LIN {X 0,Y 352.331,Z 241.453,A -85,B 0,C 180,E1 -13962.527,E2 -13962.527} C_VEL
LIN {X 0,Y 350.623,Z 232.69,A -85,B 0,C 180,E1 -13963.253,E2 -13963.253} C_VEL
LIN {X 0,Y 348.082,Z 222.748,A -85,B 0,C 180,E1 -13963.879,E2 -13963.879} C_VEL
LIN {X 0,Y 347.635,Z 220.997,A -85,B 0,C 180,E1 -13963.975,E2 -13963.975} C_VEL
LIN {X 0,Y 347.641,Z 215.336,A -85,B 0,C 180,E1 -13968.164,E2 -13968.164} C_VEL
LIN {X 0,Y 347.657,Z 211.071,A -85,B 0,C 180,E1 -13971.579,E2 -13971.579} C_VEL
LIN {X 0,Y 347.751,Z 206.902,A -85,B 0,C 180,E1 -13975.111,E2 -13975.111} C_VEL
LIN {X 0,Y 347.823,Z 203.937,A -85,B 0,C 180,E1 -13977.691,E2 -13977.691} C_VEL
LIN {X 0,Y 347.727,Z 200.189,A -85,B 0,C 180,E1 -13981.063,E2 -13981.063} C_VEL
LIN {X 0,Y 347.74,Z 200.17,A -85,B 0,C 180,E1 -13984.462,E2 -13984.462} C_VEL
LIN {X 0,Y 347.772,Z 200.165,A -85,B 0,C 180,E1 -13987.988,E2 -13987.988} C_VEL
LIN {X 0,Y 347.755,Z 200.167,A -85,B 0,C 180,E1 -13988.297,E2 -13988.297} C_VEL
LIN {X 0,Y 347.064,Z 200.255,A -85,B 0,C 180,E1 -13989.264,E2 -13989.264} C_VEL
LIN {X 0,Y 344.19,Z 200.615,A -85,B 0,C 180,E1 -13990.836,E2 -13990.836} C_VEL
LIN {X 0,Y 341.77,Z 200.915,A -85,B 0,C 180,E1 -13992.109,E2 -13992.109} C_VEL
LIN {X 0,Y 340.737,Z 201.042,A -85,B 0,C 180,E1 -13993.094,E2 -13993.094} C_VEL
LIN {X 0,Y 340.655,Z 201.049,A -85,B 0,C 180,E1 -13993.428,E2 -13993.428} C_VEL
LIN {X 0,Y 340.67,Z 201.049,A -85,B 0,C 180,E1 -13997.094,E2 -13997.094} C_VEL
LIN {X 0,Y 340.691,Z 201.044,A -85,B 0,C 180,E1 -14000.246,E2 -14000.246} C_VEL
LIN {X 0,Y 340.702,Z 201.043,A -85,B 0,C 180,E1 -14003.558,E2 -14003.558} C_VEL
LIN {X 0,Y 340.686,Z 201.043,A -85,B 0,C 180,E1 -14006.152,E2 -14006.152} C_VEL
LIN {X 0,Y 340.766,Z 201.031,A -85,B 0,C 180,E1 -14010.331,E2 -14010.331} C_VEL
LIN {X 0,Y 340.796,Z 201.032,A -85,B 0,C 180,E1 -14013.019,E2 -14013.019} C_VEL
LIN {X 0,Y 340.719,Z 201.042,A -85,B 0,C 180,E1 -14016.926,E2 -14016.926} C_VEL
LIN {X 0,Y 340.784,Z 201.03,A -85,B 0,C 180,E1 -14020.733,E2 -14020.733} C_VEL
LIN {X 0,Y 340.778,Z 201.036,A -85,B 0,C 180,E1 -14023.218,E2 -14023.218} C_VEL
LIN {X 0,Y 340.833,Z 201.027,A -85,B 0,C 180,E1 -14026.89,E2 -14026.89} C_VEL
LIN {X 0,Y 340.903,Z 201.01,A -85,B 0,C 180,E1 -14030.507,E2 -14030.507} C_VEL
LIN {X 0,Y 341.047,Z 201.002,A -85,B 0,C 180,E1 -14032.898,E2 -14032.898} C_VEL
LIN {X 0,Y 341.158,Z 200.987,A -85,B 0,C 180,E1 -14037.639,E2 -14037.639} C_VEL
LIN {X 0,Y 341.284,Z 200.96,A -85,B 0,C 180,E1 -14040,E2 -14040} C_VEL
LIN {X 0,Y 341.154,Z 200.988,A -85,B 0,C 180,E1 -14042.361,E2 -14042.361} C_VEL
LIN {X 0,Y 341.063,Z 201.001,A -85,B 0,C 180,E1 -14047.102,E2 -14047.102} C_VEL
LIN {X 0,Y 340.859,Z 201.026,A -85,B 0,C 180,E1 -14050.694,E2 -14050.694} C_VEL
LIN {X 0,Y 340.852,Z 201.022,A -85,B 0,C 180,E1 -14054.325,E2 -14054.325} C_VEL
LIN {X 0,Y 340.774,Z 201.035,A -85,B 0,C 180,E1 -14058.441,E2 -14058.441} C_VEL
LIN {X 0,Y 340.707,Z 201.048,A -85,B 0,C 180,E1 -14061.842,E2 -14061.842} C_VEL
LIN {X 0,Y 340.697,Z 201.047,A -85,B 0,C 180,E1 -14064.823,E2 -14064.823} C_VEL
LIN {X 0,Y 340.668,Z 201.051,A -85,B 0,C 180,E1 -14068.326,E2 -14068.326} C_VEL
LIN {X 0,Y 340.683,Z 201.048,A -85,B 0,C 180,E1 -14071.046,E2 -14071.046} C_VEL
LIN {X 0,Y 340.708,Z 201.043,A -85,B 0,C 180,E1 -14075.28,E2 -14075.28} C_VEL
LIN {X 0,Y 340.685,Z 201.052,A -85,B 0,C 180,E1 -14078.384,E2 -14078.384} C_VEL
LIN {X 0,Y 340.685,Z 201.044,A -85,B 0,C 180,E1 -14082.046,E2 -14082.046} C_VEL
LIN {X 0,Y 340.68,Z 201.175,A -85,B 0,C 180,E1 -14085.897,E2 -14085.897} C_VEL
LIN {X 0,Y 342.799,Z 209.575,A -85,B 0,C 180,E1 -14089.338,E2 -14089.338} C_VEL
LIN {X 0,Y 344.82,Z 218.429,A -85,B 0,C 180,E1 -14092.645,E2 -14092.645} C_VEL
LIN {X 0,Y 347.076,Z 228.6,A -85,B 0,C 180,E1 -14096.121,E2 -14096.121} C_VEL
LIN {X 0,Y 347.91,Z 233.205,A -85,B 0,C 180,E1 -14097.601,E2 -14097.601} C_VEL
LIN {X 0,Y 346.924,Z 238.889,A -85,B 0,C 180,E1 -14099.237,E2 -14099.237} C_VEL
LIN {X 0,Y 344.44,Z 253.402,A -85,B 0,C 180,E1 -14103.329,E2 -14103.329} C_VEL
LIN {X 0,Y 342.312,Z 268.107,A -85,B 0,C 180,E1 -14107.502,E2 -14107.502} C_VEL
LIN {X 0,Y 341.196,Z 277.97,A -85,B 0,C 180,E1 -14110.368,E2 -14110.368} C_VEL
LIN {X 0,Y 342.243,Z 292.548,A -85,B 0,C 180,E1 -14111.027,E2 -14111.027} C_VEL
LIN {X 0,Y 343.407,Z 308.5,A -85,B 0,C 180,E1 -14111.891,E2 -14111.891} C_VEL
LIN {X 0,Y 343.691,Z 318.722,A -85,B 0,C 180,E1 -14112.601,E2 -14112.601} C_VEL
LIN {X 0,Y 342.818,Z 330.797,A -85,B 0,C 180,E1 -14113.629,E2 -14113.629} C_VEL
LIN {X 0,Y 342.054,Z 341.26,A -85,B 0,C 180,E1 -14114.757,E2 -14114.757} C_VEL
LIN {X 0,Y 341.258,Z 350.736,A -85,B 0,C 180,E1 -14115.998,E2 -14115.998} C_VEL
LIN {X 0,Y 340.555,Z 360.121,A -85,B 0,C 180,E1 -14117.487,E2 -14117.487} C_VEL
LIN {X 0,Y 339.998,Z 367.859,A -85,B 0,C 180,E1 -14118.979,E2 -14118.979} C_VEL
LIN {X 0,Y 339.63,Z 375.408,A -85,B 0,C 180,E1 -14120.773,E2 -14120.773} C_VEL
LIN {X 0,Y 339.406,Z 382.352,A -85,B 0,C 180,E1 -14122.865,E2 -14122.865} C_VEL
LIN {X 0,Y 339.385,Z 386.872,A -85,B 0,C 180,E1 -14124.655,E2 -14124.655} C_VEL
LIN {X 0,Y 339.333,Z 390.218,A -85,B 0,C 180,E1 -14126.439,E2 -14126.439} C_VEL
LIN {X 0,Y 339.477,Z 391.85,A -85,B 0,C 180,E1 -14127.629,E2 -14127.629} C_VEL
LIN {X 0,Y 339.455,Z 393.035,A -85,B 0,C 180,E1 -14128.815,E2 -14128.815} C_VEL
LIN {X 0,Y 339.465,Z 393.781,A -85,B 0,C 180,E1 -14130.002,E2 -14130.002} C_VEL
LIN {X 0,Y 339.431,Z 394.054,A -85,B 0,C 180,E1 -14131.188,E2 -14131.188} C_VEL
LIN {X 0,Y 339.304,Z 393.908,A -85,B 0,C 180,E1 -14132.376,E2 -14132.376} C_VEL
LIN {X 0,Y 339.237,Z 393.354,A -85,B 0,C 180,E1 -14133.565,E2 -14133.565} C_VEL
LIN {X 0,Y 339.247,Z 392.357,A -85,B 0,C 180,E1 -14134.755,E2 -14134.755} C_VEL
LIN {X 0,Y 339.254,Z 390.74,A -85,B 0,C 180,E1 -14136.081,E2 -14136.081} C_VEL
LIN {X 0,Y 339.527,Z 386.809,A -85,B 0,C 180,E1 -14138.333,E2 -14138.333} C_VEL
LIN {X 0,Y 339.996,Z 382.509,A -85,B 0,C 180,E1 -14140.121,E2 -14140.121} C_VEL
LIN {X 0,Y 340.904,Z 376.038,A -85,B 0,C 180,E1 -14142.201,E2 -14142.201} C_VEL
LIN {X 0,Y 342.168,Z 369.13,A -85,B 0,C 180,E1 -14143.967,E2 -14143.967} C_VEL
LIN {X 0,Y 343.508,Z 360.231,A -85,B 0,C 180,E1 -14145.843,E2 -14145.843} C_VEL
LIN {X 0,Y 345.392,Z 350.592,A -85,B 0,C 180,E1 -14147.467,E2 -14147.467} C_VEL
LIN {X 0,Y 347.337,Z 340.326,A -85,B 0,C 180,E1 -14148.891,E2 -14148.891} C_VEL
LIN {X 0,Y 349.334,Z 329.169,A -85,B 0,C 180,E1 -14150.154,E2 -14150.154} C_VEL
LIN {X 0,Y 350.729,Z 317.833,A -85,B 0,C 180,E1 -14151.248,E2 -14151.248} C_VEL
LIN {X 0,Y 351.19,Z 306.295,A -85,B 0,C 180,E1 -14152.249,E2 -14152.249} C_VEL
LIN {X 0,Y 350.711,Z 294.905,A -85,B 0,C 180,E1 -14153.165,E2 -14153.165} C_VEL
LIN {X 0,Y 348.739,Z 281.474,A -85,B 0,C 180,E1 -14154.23,E2 -14154.23} C_VEL
LIN {X 0,Y 347.15,Z 273.498,A -85,B 0,C 180,E1 -14154.921,E2 -14154.921} C_VEL
LIN {X 0,Y 347.198,Z 262.211,A -85,B 0,C 180,E1 -14156.802,E2 -14156.802} C_VEL
LIN {X 0,Y 347.688,Z 252.609,A -85,B 0,C 180,E1 -14158.691,E2 -14158.691} C_VEL
LIN {X 0,Y 348.613,Z 243.111,A -85,B 0,C 180,E1 -14160.937,E2 -14160.937} C_VEL
LIN {X 0,Y 349.588,Z 237.732,A -85,B 0,C 180,E1 -14162.397,E2 -14162.397} C_VEL
LIN {X 0,Y 349.546,Z 234.152,A -85,B 0,C 180,E1 -14163.825,E2 -14163.825} C_VEL
LIN {X 0,Y 349.477,Z 229.371,A -85,B 0,C 180,E1 -14166.447,E2 -14166.447} C_VEL
LIN {X 0,Y 349.799,Z 226.835,A -85,B 0,C 180,E1 -14168.525,E2 -14168.525} C_VEL
LIN {X 0,Y 350.07,Z 225.471,A -85,B 0,C 180,E1 -14170.28,E2 -14170.28} C_VEL
LIN {X 0,Y 349.804,Z 225.161,A -85,B 0,C 180,E1 -14171.98,E2 -14171.98} C_VEL
LIN {X 0,Y 349.534,Z 225.849,A -85,B 0,C 180,E1 -14174.729,E2 -14174.729} C_VEL
LIN {X 0,Y 349.427,Z 227.015,A -85,B 0,C 180,E1 -14176.855,E2 -14176.855} C_VEL
LIN {X 0,Y 349.518,Z 229.704,A -85,B 0,C 180,E1 -14179.828,E2 -14179.828} C_VEL
LIN {X 0,Y 349.59,Z 233.455,A -85,B 0,C 180,E1 -14182.907,E2 -14182.907} C_VEL
LIN {X 0,Y 349.12,Z 235.637,A -85,B 0,C 180,E1 -14184.282,E2 -14184.282} C_VEL
LIN {X 0,Y 347.059,Z 244.028,A -85,B 0,C 180,E1 -14188.91,E2 -14188.91} C_VEL
LIN {X 0,Y 345.791,Z 251.511,A -85,B 0,C 180,E1 -14192.787,E2 -14192.787} C_VEL
LIN {X 0,Y 345.214,Z 255.87,A -85,B 0,C 180,E1 -14194.979,E2 -14194.979} C_VEL
LIN {X 0,Y 350.216,Z 269.193,A -85,B 0,C 180,E1 -14196.642,E2 -14196.642} C_VEL
LIN {X 0,Y 352.966,Z 279.492,A -85,B 0,C 180,E1 -14197.88,E2 -14197.88} C_VEL
LIN {X 0,Y 353.856,Z 284.485,A -85,B 0,C 180,E1 -14198.471,E2 -14198.471} C_VEL
LIN {X 0,Y 353.542,Z 288.493,A -85,B 0,C 180,E1 -14198.84,E2 -14198.84} C_VEL
LIN {X 0,Y 351.506,Z 301.336,A -85,B 0,C 180,E1 -14200.129,E2 -14200.129} C_VEL
LIN {X 0,Y 349.481,Z 312.503,A -85,B 0,C 180,E1 -14201.535,E2 -14201.535} C_VEL
LIN {X 0,Y 347.312,Z 323.385,A -85,B 0,C 180,E1 -14203.241,E2 -14203.241} C_VEL
LIN {X 0,Y 345.426,Z 332.168,A -85,B 0,C 180,E1 -14204.965,E2 -14204.965} C_VEL
LIN {X 0,Y 343.877,Z 339.374,A -85,B 0,C 180,E1 -14206.707,E2 -14206.707} C_VEL
LIN {X 0,Y 342.49,Z 346.013,A -85,B 0,C 180,E1 -14208.759,E2 -14208.759} C_VEL
LIN {X 0,Y 341.516,Z 350.471,A -85,B 0,C 180,E1 -14210.524,E2 -14210.524} C_VEL
LIN {X 0,Y 340.957,Z 352.869,A -85,B 0,C 180,E1 -14211.704,E2 -14211.704} C_VEL
LIN {X 0,Y 340.36,Z 354.823,A -85,B 0,C 180,E1 -14212.883,E2 -14212.883} C_VEL
LIN {X 0,Y 340.03,Z 357.387,A -85,B 0,C 180,E1 -14215.258,E2 -14215.258} C_VEL
LIN {X 0,Y 339.77,Z 358.097,A -85,B 0,C 180,E1 -14216.442,E2 -14216.442} C_VEL
LIN {X 0,Y 339.543,Z 358.363,A -85,B 0,C 180,E1 -14217.628,E2 -14217.628} C_VEL
LIN {X 0,Y 339.394,Z 358.233,A -85,B 0,C 180,E1 -14218.814,E2 -14218.814} C_VEL
LIN {X 0,Y 339.313,Z 357.708,A -85,B 0,C 180,E1 -14220,E2 -14220} C_VEL
LIN {X 0,Y 339.288,Z 356.746,A -85,B 0,C 180,E1 -14221.187,E2 -14221.187} C_VEL
LIN {X 0,Y 339.285,Z 355.356,A -85,B 0,C 180,E1 -14222.374,E2 -14222.374} C_VEL
LIN {X 0,Y 339.386,Z 352.47,A -85,B 0,C 180,E1 -14224.156,E2 -14224.156} C_VEL
LIN {X 0,Y 339.531,Z 348.538,A -85,B 0,C 180,E1 -14225.941,E2 -14225.941} C_VEL
LIN {X 0,Y 339.828,Z 343.458,A -85,B 0,C 180,E1 -14227.726,E2 -14227.726} C_VEL
LIN {X 0,Y 340.3,Z 337.094,A -85,B 0,C 180,E1 -14229.51,E2 -14229.51} C_VEL
LIN {X 0,Y 340.92,Z 329.168,A -85,B 0,C 180,E1 -14231.294,E2 -14231.294} C_VEL
LIN {X 0,Y 341.705,Z 319.396,A -85,B 0,C 180,E1 -14233.076,E2 -14233.076} C_VEL
LIN {X 0,Y 342.518,Z 309.344,A -85,B 0,C 180,E1 -14234.558,E2 -14234.558} C_VEL
LIN {X 0,Y 343.369,Z 298.225,A -85,B 0,C 180,E1 -14235.899,E2 -14235.899} C_VEL
LIN {X 0,Y 344.234,Z 286.092,A -85,B 0,C 180,E1 -14237.067,E2 -14237.067} C_VEL
LIN {X 0,Y 344.912,Z 275.241,A -85,B 0,C 180,E1 -14237.897,E2 -14237.897} C_VEL
LIN {X 0,Y 342.797,Z 261.842,A -85,B 0,C 180,E1 -14238.779,E2 -14238.779} C_VEL
